	W =  -167.362 deg,	P =    -0.001 deg,	R =   120.301 deg
};
P[2889]{
   GP1:
	UF : 7, UT : 3,	CONFIG : 'F U T, 0, 0, 0',
	X =   278.445  mm,	Y =    78.332  mm,	Z =     0.000  mm,
	W =  -167.362 deg,	P =    -0.001 deg,	R =   120.301 deg
};
P[2890]{
   GP1:
	UF : 7, UT : 3,	CONFIG : 'F U T, 0, 0, 0',
	X =   278.445  mm,	Y =    78.332  mm,	Z =     0.000  mm,
	W =  -167.362 deg,	P =    -0.001 deg,	R =   120.301 deg
};
P[2891]{
   GP1:
	UF : 7, UT : 3,	CONFIG : 'F U T, 0, 0, 0',
	X =   278.445  mm,	Y =    78.332  mm,	Z =     0.000  mm,
	W =  -167.362 deg,	P =    -0.001 deg,	R =   120.301 deg
};
P[2892]{
   GP1:
	UF : 7, UT : 3,	CONFIG : 'F U T, 0, 0, 0',
	X =   272.605  mm,	Y =    96.720  mm,	Z =     0.001  mm,
	W =  -167.361 deg,	P =    -0.001 deg,	R =   124.584 deg
};
P[2893]{
   GP1:
	UF : 7, UT : 3,	CONFIG : 'F U T, 0, 0, 0',
	X =   265.154  mm,	Y =   115.600  mm,	Z =     0.001  mm,
	W =  -167.361 deg,	P =     0.000 deg,	R =   128.604 deg
};
P[2894]{
   GP1:
	UF : 7, UT : 3,	CONFIG : 'F U T, 0, 0, 0',
	X =   256.399  mm,	Y =   133.902  mm,	Z =     0.002  mm,
	W =  -167.361 deg,	P =     0.000 deg,	R =   132.625 deg
};
P[2895]{
   GP1:
	UF : 7, UT : 3,	CONFIG : 'F U T, 0, 0, 0',
	X =   246.387  mm,	Y =   151.536  mm,	Z =     0.001  mm,
	W =  -167.360 deg,	P =     0.000 deg,	R =   136.648 deg
};
P[2896]{
   GP1:
	UF : 7, UT : 3,	CONFIG : 'F U T, 0, 0, 0',
	X =   234.864  mm,	Y =   168.850  mm,	Z =     0.000  mm,
	W =  -167.359 deg,	P =     0.001 deg,	R =   140.583 deg
};
P[2897]{
   GP1:
	UF : 7, UT : 3,	CONFIG : 'F U T, 0, 0, 0',
	X =   234.864  mm,	Y =   168.850  mm,	Z =     0.000  mm,
	W =  -167.359 deg,	P =     0.001 deg,	R =   140.583 deg
};
P[2898]{
   GP1:
	UF : 7, UT : 3,	CONFIG : 'F U T, 0, 0, 0',
	X =   234.864  mm,	Y =   168.850  mm,	Z =     0.000  mm,
	W =  -167.359 deg,	P =     0.001 deg,	R =   140.583 deg
};
P[2899]{
   GP1:
	UF : 7, UT : 3,	CONFIG : 'F U T, 0, 0, 0',
	X =   234.864  mm,	Y =   168.850  mm,	Z =     0.000  mm,
	W =  -167.359 deg,	P =     0.001 deg,	R =   140.583 deg
};
P[2900]{
   GP1:
	UF : 7, UT : 3,	CONFIG : 'F U T, 0, 0, 0',
	X =   216.882  mm,	Y =   191.391  mm,	Z =     0.000  mm,
	W =  -167.361 deg,	P =    -0.002 deg,	R =   146.469 deg
};
P[2901]{
   GP1:
	UF : 7, UT : 3,	CONFIG : 'F U T, 0, 0, 0',
	X =   216.882  mm,	Y =   191.391  mm,	Z =     0.000  mm,
	W =  -167.361 deg,	P =    -0.002 deg,	R =   146.469 deg
};
P[2902]{
   GP1:
	UF : 7, UT : 3,	CONFIG : 'F U T, 0, 0, 0',
	X =   216.882  mm,	Y =   191.391  mm,	Z =     0.000  mm,
	W =  -167.361 deg,	P =    -0.002 deg,	R =   146.469 deg
};
P[2903]{
   GP1:
	UF : 7, UT : 3,	CONFIG : 'F U T, 0, 0, 0',
	X =   216.882  mm,	Y =   191.391  mm,	Z =     0.000  mm,
	W =  -167.361 deg,	P =    -0.002 deg,	R =   146.469 deg
};
P[2904]{
   GP1:
	UF : 7, UT : 3,	CONFIG : 'F U T, 0, 0, 0',
	X =   203.003  mm,	Y =   206.059  mm,	Z =     0.001  mm,
	W =  -167.361 deg,	P =    -0.002 deg,	R =   150.475 deg
};
P[2905]{
   GP1:
	UF : 7, UT : 3,	CONFIG : 'F U T, 0, 0, 0',
	X =   188.133  mm,	Y =   219.721  mm,	Z =     0.001  mm,
	W =  -167.360 deg,	P =    -0.001 deg,	R =   154.481 deg
};
P[2906]{
   GP1:
	UF : 7, UT : 3,	CONFIG : 'F U T, 0, 0, 0',
	X =   172.345  mm,	Y =   232.311  mm,	Z =     0.001  mm,
	W =  -167.360 deg,	P =     0.000 deg,	R =   158.487 deg
};
P[2907]{
   GP1:
	UF : 7, UT : 3,	CONFIG : 'F U T, 0, 0, 0',
	X =   155.715  mm,	Y =   243.767  mm,	Z =     0.001  mm,
	W =  -167.359 deg,	P =     0.000 deg,	R =   162.492 deg
};
P[2908]{
   GP1:
	UF : 7, UT : 3,	CONFIG : 'F U T, 0, 0, 0',
	X =   138.327  mm,	Y =   254.033  mm,	Z =     0.000  mm,
	W =  -167.359 deg,	P =     0.001 deg,	R =   166.498 deg
};
P[2909]{
   GP1:
	UF : 7, UT : 3,	CONFIG : 'F U T, 0, 0, 0',
	X =   138.327  mm,	Y =   254.033  mm,	Z =     0.000  mm,
	W =  -167.359 deg,	P =     0.001 deg,	R =   166.498 deg
};
P[2910]{
   GP1:
	UF : 7, UT : 3,	CONFIG : 'F U T, 0, 0, 0',
	X =   138.327  mm,	Y =   254.033  mm,	Z =     0.000  mm,
	W =  -167.359 deg,	P =     0.001 deg,	R =   166.498 deg
};
P[2911]{
   GP1:
	UF : 7, UT : 3,	CONFIG : 'F U T, 0, 0, 0',
	X =   138.327  mm,	Y =   254.033  mm,	Z =     0.000  mm,
	W =  -167.359 deg,	P =     0.001 deg,	R =   166.498 deg
};
P[2912]{
   GP1:
	UF : 7, UT : 3,	CONFIG : 'F U T, 0, 0, 0',
	X =   112.342  mm,	Y =   266.562  mm,	Z =     0.000  mm,
	W =  -167.361 deg,	P =    -0.002 deg,	R =   172.748 deg
};
P[2913]{
   GP1:
	UF : 7, UT : 3,	CONFIG : 'F U T, 0, 0, 0',
	X =   112.342  mm,	Y =   266.562  mm,	Z =     0.000  mm,
	W =  -167.361 deg,	P =    -0.002 deg,	R =   172.748 deg
};
P[2914]{
   GP1:
	UF : 7, UT : 3,	CONFIG : 'F U T, 0, 0, 0',
	X =   112.342  mm,	Y =   266.562  mm,	Z =     0.000  mm,
	W =  -167.361 deg,	P =    -0.002 deg,	R =   172.748 deg
};
P[2915]{
   GP1:
	UF : 7, UT : 3,	CONFIG : 'F U T, 0, 0, 0',
	X =   112.342  mm,	Y =   266.562  mm,	Z =     0.000  mm,
	W =  -167.361 deg,	P =    -0.002 deg,	R =   172.748 deg
};
P[2916]{
   GP1:
	UF : 7, UT : 3,	CONFIG : 'F U T, 0, 0, 0',
	X =    91.881  mm,	Y =   274.273  mm,	Z =     0.001  mm,
	W =  -167.361 deg,	P =    -0.001 deg,	R =   176.495 deg
};
P[2917]{
   GP1:
	UF : 7, UT : 3,	CONFIG : 'F U T, 0, 0, 0',
	X =    72.938  mm,	Y =   279.908  mm,	Z =     0.001  mm,
	W =  -167.361 deg,	P =    -0.001 deg,	R =  -179.569 deg
};
P[2918]{
   GP1:
	UF : 7, UT : 3,	CONFIG : 'F U T, 0, 0, 0',
	X =    53.633  mm,	Y =   284.242  mm,	Z =     0.001  mm,
	W =  -167.361 deg,	P =     0.000 deg,	R =  -175.638 deg
};
P[2919]{
   GP1:
	UF : 7, UT : 3,	CONFIG : 'F U T, 0, 0, 0',
	X =    34.061  mm,	Y =   287.246  mm,	Z =     0.001  mm,
	W =  -167.360 deg,	P =     0.000 deg,	R =  -171.710 deg
};
P[2920]{
   GP1:
	UF : 7, UT : 3,	CONFIG : 'F U T, 0, 0, 0',
	X =    14.416  mm,	Y =   288.897  mm,	Z =     0.000  mm,
	W =  -167.360 deg,	P =     0.001 deg,	R =  -167.766 deg
};
P[2921]{
   GP1:
	UF : 7, UT : 3,	CONFIG : 'F U T, 0, 0, 0',
	X =    14.416  mm,	Y =   288.897  mm,	Z =     0.000  mm,
	W =  -167.360 deg,	P =     0.001 deg,	R =  -167.766 deg
};
P[2922]{
   GP1:
	UF : 7, UT : 3,	CONFIG : 'F U T, 0, 0, 0',
	X =    14.416  mm,	Y =   288.897  mm,	Z =     0.000  mm,
	W =  -167.360 deg,	P =     0.001 deg,	R =  -167.766 deg
};
P[2923]{
   GP1:
	UF : 7, UT : 3,	CONFIG : 'F U T, 0, 0, 0',
	X =    14.416  mm,	Y =   288.897  mm,	Z =     0.000  mm,
	W =  -167.360 deg,	P =     0.001 deg,	R =  -167.766 deg
};
P[2924]{
   GP1:
	UF : 7, UT : 3,	CONFIG : 'F U T, 0, 0, 0',
	X =   -14.416  mm,	Y =   288.897  mm,	Z =     0.000  mm,
	W =  -167.360 deg,	P =    -0.003 deg,	R =  -162.071 deg
};
P[2925]{
   GP1:
	UF : 7, UT : 3,	CONFIG : 'F U T, 0, 0, 0',
	X =   -14.416  mm,	Y =   288.897  mm,	Z =     0.000  mm,
	W =  -167.360 deg,	P =    -0.003 deg,	R =  -162.071 deg
};
P[2926]{
   GP1:
	UF : 7, UT : 3,	CONFIG : 'F U T, 0, 0, 0',
	X =   -14.416  mm,	Y =   288.897  mm,	Z =     0.000  mm,
	W =  -167.360 deg,	P =    -0.003 deg,	R =  -162.071 deg
};
P[2927]{
   GP1:
	UF : 7, UT : 3,	CONFIG : 'F U T, 0, 0, 0',
	X =   -14.416  mm,	Y =   288.897  mm,	Z =     0.000  mm,
	W =  -167.360 deg,	P =    -0.003 deg,	R =  -162.071 deg
};
P[2928]{
   GP1:
	UF : 7, UT : 3,	CONFIG : 'F U T, 0, 0, 0',
	X =   -34.138  mm,	Y =   287.238  mm,	Z =     0.001  mm,
	W =  -167.359 deg,	P =    -0.001 deg,	R =  -158.155 deg
};
P[2929]{
   GP1:
	UF : 7, UT : 3,	CONFIG : 'F U T, 0, 0, 0',
	X =   -53.719  mm,	Y =   284.226  mm,	Z =     0.002  mm,
	W =  -167.358 deg,	P =     0.000 deg,	R =  -154.243 deg
};
P[2930]{
   GP1:
	UF : 7, UT : 3,	CONFIG : 'F U T, 0, 0, 0',
	X =   -73.012  mm,	Y =   279.888  mm,	Z =     0.002  mm,
	W =  -167.356 deg,	P =     0.001 deg,	R =  -150.325 deg
};
P[2931]{
   GP1:
	UF : 7, UT : 3,	CONFIG : 'F U T, 0, 0, 0',
	X =   -91.931  mm,	Y =   274.255  mm,	Z =     0.002  mm,
	W =  -167.354 deg,	P =     0.002 deg,	R =  -146.400 deg
};
P[2932]{
   GP1:
	UF : 7, UT : 3,	CONFIG : 'F U T, 0, 0, 0',
	X =  -112.342  mm,	Y =   266.562  mm,	Z =     0.000  mm,
	W =  -167.352 deg,	P =     0.002 deg,	R =  -142.645 deg
};
P[2933]{
   GP1:
	UF : 7, UT : 3,	CONFIG : 'F U T, 0, 0, 0',
	X =  -112.342  mm,	Y =   266.562  mm,	Z =     0.000  mm,
	W =  -167.352 deg,	P =     0.002 deg,	R =  -142.645 deg
};
P[2934]{
   GP1:
	UF : 7, UT : 3,	CONFIG : 'F U T, 0, 0, 0',
	X =  -112.342  mm,	Y =   266.562  mm,	Z =     0.000  mm,
	W =  -167.352 deg,	P =     0.002 deg,	R =  -142.645 deg
};
P[2935]{
   GP1:
	UF : 7, UT : 3,	CONFIG : 'F U T, 0, 0, 0',
	X =  -112.342  mm,	Y =   266.562  mm,	Z =     0.000  mm,
	W =  -167.352 deg,	P =     0.002 deg,	R =  -142.645 deg
};
P[2936]{
   GP1:
	UF : 7, UT : 3,	CONFIG : 'F U T, 0, 0, 0',
	X =  -138.327  mm,	Y =   254.033  mm,	Z =     0.000  mm,
	W =  -167.342 deg,	P =    -0.019 deg,	R =  -136.890 deg
};
P[2937]{
   GP1:
	UF : 7, UT : 3,	CONFIG : 'F U T, 0, 0, 0',
	X =  -138.327  mm,	Y =   254.033  mm,	Z =     0.000  mm,
	W =  -167.342 deg,	P =    -0.019 deg,	R =  -136.890 deg
};
P[2938]{
   GP1:
	UF : 7, UT : 3,	CONFIG : 'F U T, 0, 0, 0',
	X =  -138.327  mm,	Y =   254.033  mm,	Z =     0.000  mm,
	W =  -167.342 deg,	P =    -0.019 deg,	R =  -136.890 deg
};
P[2939]{
   GP1:
	UF : 7, UT : 3,	CONFIG : 'F U T, 0, 0, 0',
	X =  -138.327  mm,	Y =   254.033  mm,	Z =     0.000  mm,
	W =  -167.342 deg,	P =    -0.019 deg,	R =  -136.890 deg
};
P[2940]{
   GP1:
	UF : 7, UT : 3,	CONFIG : 'F U T, 0, 0, 0',
	X =  -150.066  mm,	Y =   247.282  mm,	Z =     0.005  mm,
	W =  -167.352 deg,	P =    -0.024 deg,	R =  -133.674 deg
};
P[2941]{
   GP1:
	UF : 7, UT : 3,	CONFIG : 'F U T, 0, 0, 0',
	X =  -162.485  mm,	Y =   239.322  mm,	Z =     0.016  mm,
	W =  -167.364 deg,	P =    -0.028 deg,	R =  -130.774 deg
};
P[2942]{
   GP1:
	UF : 7, UT : 3,	CONFIG : 'F U T, 0, 0, 0',
	X =  -174.433  mm,	Y =   230.744  mm,	Z =     0.026  mm,
	W =  -167.376 deg,	P =    -0.032 deg,	R =  -127.865 deg
};
P[2943]{
   GP1:
	UF : 7, UT : 3,	CONFIG : 'F U T, 0, 0, 0',
	X =  -187.272  mm,	Y =   220.459  mm,	Z =     0.032  mm,
	W =  -167.361 deg,	P =     0.001 deg,	R =  -124.599 deg
};
P[2944]{
   GP1:
	UF : 7, UT : 3,	CONFIG : 'F U T, 0, 0, 0',
	X =  -199.499  mm,	Y =   209.447  mm,	Z =     0.028  mm,
	W =  -167.343 deg,	P =     0.031 deg,	R =  -121.336 deg
};
P[2945]{
   GP1:
	UF : 7, UT : 3,	CONFIG : 'F U T, 0, 0, 0',
	X =  -208.545  mm,	Y =   200.442  mm,	Z =     0.017  mm,
	W =  -167.261 deg,	P =     0.037 deg,	R =  -118.804 deg
};
P[2946]{
   GP1:
	UF : 7, UT : 3,	CONFIG : 'F U T, 0, 0, 0',
	X =  -216.882  mm,	Y =   191.391  mm,	Z =     0.000  mm,
	W =  -167.182 deg,	P =     0.034 deg,	R =  -116.167 deg
};
P[2947]{
   GP1:
	UF : 7, UT : 3,	CONFIG : 'F U T, 0, 0, 0',
	X =  -216.882  mm,	Y =   191.391  mm,	Z =     0.000  mm,
	W =  -167.182 deg,	P =     0.034 deg,	R =  -116.167 deg
};
P[2948]{
   GP1:
	UF : 7, UT : 3,	CONFIG : 'F U T, 0, 0, 0',
	X =  -216.882  mm,	Y =   191.391  mm,	Z =     0.000  mm,
	W =  -167.182 deg,	P =     0.034 deg,	R =  -116.167 deg
};
P[2949]{
   GP1:
	UF : 7, UT : 3,	CONFIG : 'F U T, 0, 0, 0',
	X =  -216.882  mm,	Y =   191.391  mm,	Z =     0.000  mm,
	W =  -167.182 deg,	P =     0.034 deg,	R =  -116.167 deg
};
P[2950]{
   GP1:
	UF : 7, UT : 3,	CONFIG : 'F U T, 0, 0, 0',
	X =  -234.864  mm,	Y =   168.850  mm,	Z =     0.000  mm,
	W =  -167.097 deg,	P =    -0.235 deg,	R =  -110.476 deg
};
P[2951]{
   GP1:
	UF : 7, UT : 3,	CONFIG : 'F U T, 0, 0, 0',
	X =  -234.864  mm,	Y =   168.850  mm,	Z =     0.000  mm,
	W =  -167.097 deg,	P =    -0.235 deg,	R =  -110.476 deg
};
P[2952]{
   GP1:
	UF : 7, UT : 3,	CONFIG : 'F U T, 0, 0, 0',
	X =  -234.864  mm,	Y =   168.850  mm,	Z =     0.000  mm,
	W =  -167.097 deg,	P =    -0.235 deg,	R =  -110.476 deg
};
P[2953]{
   GP1:
	UF : 7, UT : 3,	CONFIG : 'F U T, 0, 0, 0',
	X =  -234.864  mm,	Y =   168.850  mm,	Z =     0.000  mm,
	W =  -167.097 deg,	P =    -0.235 deg,	R =  -110.476 deg
};
P[2954]{
   GP1:
	UF : 7, UT : 3,	CONFIG : 'F U T, 0, 0, 0',
	X =  -241.066  mm,	Y =   159.864  mm,	Z =     0.043  mm,
	W =  -167.290 deg,	P =    -0.308 deg,	R =  -108.496 deg
};
P[2955]{
   GP1:
	UF : 7, UT : 3,	CONFIG : 'F U T, 0, 0, 0',
	X =  -248.977  mm,	Y =   147.242  mm,	Z =     0.116  mm,
	W =  -167.654 deg,	P =    -0.189 deg,	R =  -105.549 deg
};
P[2956]{
   GP1:
	UF : 7, UT : 3,	CONFIG : 'F U T, 0, 0, 0',
	X =  -255.396  mm,	Y =   135.803  mm,	Z =     0.159  mm,
	W =  -167.849 deg,	P =     0.033 deg,	R =  -102.948 deg
};
P[2957]{
   GP1:
	UF : 7, UT : 3,	CONFIG : 'F U T, 0, 0, 0',
	X =  -260.804  mm,	Y =   125.101  mm,	Z =     0.156  mm,
	W =  -167.842 deg,	P =     0.260 deg,	R =  -100.577 deg
};
P[2958]{
   GP1:
	UF : 7, UT : 3,	CONFIG : 'F U T, 0, 0, 0',
	X =  -269.129  mm,	Y =   106.023  mm,	Z =     0.064  mm,
	W =  -167.476 deg,	P =     0.308 deg,	R =   -96.448 deg
};
P[2959]{
   GP1:
	UF : 7, UT : 3,	CONFIG : 'F U T, 0, 0, 0',
	X =  -273.782  mm,	Y =    93.358  mm,	Z =     0.017  mm,
	W =  -167.326 deg,	P =     0.122 deg,	R =   -93.774 deg
};
P[2960]{
   GP1:
	UF : 7, UT : 3,	CONFIG : 'F U T, 0, 0, 0',
	X =  -278.445  mm,	Y =    78.332  mm,	Z =     0.000  mm,
	W =  -167.321 deg,	P =     0.009 deg,	R =   -90.279 deg
};
P[2961]{
   GP1:
	UF : 7, UT : 3,	CONFIG : 'F U T, 0, 0, 0',
	X =  -278.445  mm,	Y =    78.332  mm,	Z =     0.000  mm,
	W =  -167.321 deg,	P =     0.009 deg,	R =   -90.279 deg
};
P[2962]{
   GP1:
	UF : 7, UT : 3,	CONFIG : 'F U T, 0, 0, 0',
	X =  -278.445  mm,	Y =    78.332  mm,	Z =     0.000  mm,
	W =  -167.321 deg,	P =     0.009 deg,	R =   -90.279 deg
};
P[2963]{
   GP1:
	UF : 7, UT : 3,	CONFIG : 'F U T, 0, 0, 0',
	X =  -278.445  mm,	Y =    78.332  mm,	Z =     0.000  mm,
	W =  -167.321 deg,	P =     0.009 deg,	R =   -90.279 deg
};
P[2964]{
   GP1:
	UF : 7, UT : 3,	CONFIG : 'F U T, 0, 1, 0',
	X =  -284.871  mm,	Y =    50.219  mm,	Z =     0.000  mm,
	W =  -167.355 deg,	P =    -0.008 deg,	R =   -84.578 deg
};
P[2965]{
   GP1:
	UF : 7, UT : 3,	CONFIG : 'F U T, 0, 1, 0',
	X =  -284.871  mm,	Y =    50.219  mm,	Z =     0.000  mm,
	W =  -167.355 deg,	P =    -0.008 deg,	R =   -84.578 deg
};
P[2966]{
   GP1:
	UF : 7, UT : 3,	CONFIG : 'F U T, 0, 1, 0',
	X =  -284.871  mm,	Y =    50.219  mm,	Z =     0.000  mm,
	W =  -167.355 deg,	P =    -0.008 deg,	R =   -84.578 deg
};
P[2967]{
   GP1:
	UF : 7, UT : 3,	CONFIG : 'F U T, 0, 1, 0',
	X =  -284.871  mm,	Y =    50.219  mm,	Z =     0.000  mm,
	W =  -167.355 deg,	P =    -0.008 deg,	R =   -84.578 deg
};
P[2968]{
   GP1:
	UF : 7, UT : 3,	CONFIG : 'F U T, 0, 1, 0',
	X =  -287.321  mm,	Y =    33.420  mm,	Z =     0.001  mm,
	W =  -167.358 deg,	P =    -0.004 deg,	R =   -81.599 deg
};
P[2969]{
   GP1:
	UF : 7, UT : 3,	CONFIG : 'F U T, 0, 1, 0',
	X =  -288.718  mm,	Y =    17.699  mm,	Z =     0.001  mm,
	W =  -167.360 deg,	P =     0.000 deg,	R =   -78.468 deg
};
P[2970]{
   GP1:
	UF : 7, UT : 3,	CONFIG : 'F U T, 0, 1, 0',
	X =  -289.270  mm,	Y =     0.000  mm,	Z =     0.000  mm,
	W =  -167.362 deg,	P =     0.004 deg,	R =   -75.519 deg
};
P[2971]{
   GP1:
	UF : 7, UT : 3,	CONFIG : 'F U T, 0, 1, 0',
	X =  -289.270  mm,	Y =     0.000  mm,	Z =     0.000  mm,
	W =  -167.362 deg,	P =     0.004 deg,	R =   -75.519 deg
};
P[2972]{
   GP1:
	UF : 7, UT : 3,	CONFIG : 'F U T, 0, 1, 0',
	X =  -289.270  mm,	Y =     0.000  mm,	Z =     0.000  mm,
	W =  -167.362 deg,	P =     0.004 deg,	R =   -75.519 deg
};
P[2973]{
   GP1:
	UF : 7, UT : 3,	CONFIG : 'F U T, 0, 1, 0',
	X =  -289.270  mm,	Y =     0.000  mm,	Z =     0.000  mm,
	W =  -167.362 deg,	P =     0.004 deg,	R =   -75.519 deg
};
P[2974]{
   GP1:
	UF : 7, UT : 3,	CONFIG : 'F U T, 0, 1, 0',
	X =  -286.136  mm,	Y =     0.000  mm,	Z =     0.000  mm,
	W =  -167.363 deg,	P =     0.004 deg,	R =   -75.540 deg
};
P[2975]{
   GP1:
	UF : 7, UT : 3,	CONFIG : 'F U T, 0, 1, 0',
	X =  -286.136  mm,	Y =     0.000  mm,	Z =     0.000  mm,
	W =  -167.363 deg,	P =     0.004 deg,	R =   -75.540 deg
};
P[2976]{
   GP1:
	UF : 7, UT : 3,	CONFIG : 'F U T, 0, 1, 0',
	X =  -286.136  mm,	Y =     0.000  mm,	Z =     0.000  mm,
	W =  -167.363 deg,	P =     0.004 deg,	R =   -75.540 deg
};
P[2977]{
   GP1:
	UF : 7, UT : 3,	CONFIG : 'F U T, 0, 1, 0',
	X =  -286.136  mm,	Y =     0.000  mm,	Z =     0.000  mm,
	W =  -167.363 deg,	P =     0.004 deg,	R =   -75.540 deg
};
P[2978]{
   GP1:
	UF : 7, UT : 3,	CONFIG : 'F U T, 0, 1, 0',
	X =  -285.285  mm,	Y =    21.849  mm,	Z =     0.001  mm,
	W =  -167.358 deg,	P =     0.000 deg,	R =   -79.336 deg
};
P[2979]{
   GP1:
	UF : 7, UT : 3,	CONFIG : 'F U T, 0, 1, 0',
	X =  -283.088  mm,	Y =    41.562  mm,	Z =     0.001  mm,
	W =  -167.354 deg,	P =    -0.003 deg,	R =   -83.290 deg
};
P[2980]{
   GP1:
	UF : 7, UT : 3,	CONFIG : 'F U T, 0, 0, 0',
	X =  -279.677  mm,	Y =    60.374  mm,	Z =     0.000  mm,
	W =  -167.350 deg,	P =    -0.005 deg,	R =   -87.604 deg
};
P[2981]{
   GP1:
	UF : 7, UT : 3,	CONFIG : 'F U T, 0, 0, 0',
	X =  -275.294  mm,	Y =    77.973  mm,	Z =     0.002  mm,
	W =  -167.340 deg,	P =     0.036 deg,	R =   -90.757 deg
};
P[2982]{
   GP1:
	UF : 7, UT : 3,	CONFIG : 'F U T, 0, 0, 0',
	X =  -271.856  mm,	Y =    89.226  mm,	Z =     0.011  mm,
	W =  -167.339 deg,	P =     0.076 deg,	R =   -93.116 deg
};
P[2983]{
   GP1:
	UF : 7, UT : 3,	CONFIG : 'F U T, 0, 0, 0',
	X =  -266.629  mm,	Y =   103.805  mm,	Z =     0.050  mm,
	W =  -167.469 deg,	P =     0.237 deg,	R =   -96.222 deg
};
P[2984]{
   GP1:
	UF : 7, UT : 3,	CONFIG : 'F U T, 0, 0, 0',
	X =  -261.798  mm,	Y =   115.450  mm,	Z =     0.101  mm,
	W =  -167.689 deg,	P =     0.319 deg,	R =   -98.743 deg
};
P[2985]{
   GP1:
	UF : 7, UT : 3,	CONFIG : 'F U T, 0, 0, 0',
	X =  -256.793  mm,	Y =   126.192  mm,	Z =     0.132  mm,
	W =  -167.832 deg,	P =     0.202 deg,	R =  -101.119 deg
};
P[2986]{
   GP1:
	UF : 7, UT : 3,	CONFIG : 'F U T, 0, 0, 0',
	X =  -250.756  mm,	Y =   137.801  mm,	Z =     0.128  mm,
	W =  -167.798 deg,	P =     0.001 deg,	R =  -103.739 deg
};
P[2987]{
   GP1:
	UF : 7, UT : 3,	CONFIG : 'F U T, 0, 0, 0',
	X =  -242.629  mm,	Y =   151.646  mm,	Z =     0.077  mm,
	W =  -167.535 deg,	P =    -0.178 deg,	R =  -106.947 deg
};
P[2988]{
   GP1:
	UF : 7, UT : 3,	CONFIG : 'F U T, 0, 0, 0',
	X =  -233.847  mm,	Y =   164.876  mm,	Z =     0.022  mm,
	W =  -167.222 deg,	P =    -0.201 deg,	R =  -110.133 deg
};
P[2989]{
   GP1:
	UF : 7, UT : 3,	CONFIG : 'F U T, 0, 0, 0',
	X =  -221.510  mm,	Y =   181.125  mm,	Z =     0.000  mm,
	W =  -167.152 deg,	P =    -0.034 deg,	R =  -114.137 deg
};
P[2990]{
   GP1:
	UF : 7, UT : 3,	CONFIG : 'F U T, 0, 0, 0',
	X =  -207.946  mm,	Y =   196.530  mm,	Z =     0.018  mm,
	W =  -167.290 deg,	P =     0.036 deg,	R =  -118.342 deg
};
P[2991]{
   GP1:
	UF : 7, UT : 3,	CONFIG : 'F U T, 0, 0, 0',
	X =  -198.736  mm,	Y =   205.842  mm,	Z =     0.028  mm,
	W =  -167.341 deg,	P =     0.025 deg,	R =  -120.961 deg
};
P[2992]{
   GP1:
	UF : 7, UT : 3,	CONFIG : 'F U T, 0, 0, 0',
	X =  -189.097  mm,	Y =   214.731  mm,	Z =     0.031  mm,
	W =  -167.391 deg,	P =     0.010 deg,	R =  -123.576 deg
};
P[2993]{
   GP1:
	UF : 7, UT : 3,	CONFIG : 'F U T, 0, 0, 0',
	X =  -174.298  mm,	Y =   226.904  mm,	Z =     0.027  mm,
	W =  -167.380 deg,	P =    -0.016 deg,	R =  -127.397 deg
};
P[2994]{
   GP1:
	UF : 7, UT : 3,	CONFIG : 'F U T, 0, 0, 0',
	X =  -158.838  mm,	Y =   237.981  mm,	Z =     0.015  mm,
	W =  -167.365 deg,	P =    -0.041 deg,	R =  -131.246 deg
};
P[2995]{
   GP1:
	UF : 7, UT : 3,	CONFIG : 'F U T, 0, 0, 0',
	X =  -143.540  mm,	Y =   247.511  mm,	Z =     0.004  mm,
	W =  -167.354 deg,	P =    -0.025 deg,	R =  -134.853 deg
};
P[2996]{
   GP1:
	UF : 7, UT : 3,	CONFIG : 'F U T, 0, 0, 0',
	X =  -127.238  mm,	Y =   256.279  mm,	Z =     0.000  mm,
	W =  -167.345 deg,	P =    -0.007 deg,	R =  -138.815 deg
};
P[2997]{
   GP1:
	UF : 7, UT : 3,	CONFIG : 'F U T, 0, 0, 0',
	X =  -121.064  mm,	Y =   259.248  mm,	Z =     0.000  mm,
	W =  -167.348 deg,	P =    -0.003 deg,	R =  -139.601 deg
};
P[2998]{
   GP1:
	UF : 7, UT : 3,	CONFIG : 'F U T, 0, 0, 0',
	X =  -102.132  mm,	Y =   267.271  mm,	Z =     0.001  mm,
	W =  -167.350 deg,	P =    -0.002 deg,	R =  -144.019 deg
};
P[2999]{
   GP1:
	UF : 7, UT : 3,	CONFIG : 'F U T, 0, 0, 0',
	X =   -82.792  mm,	Y =   273.885  mm,	Z =     0.002  mm,
	W =  -167.352 deg,	P =    -0.001 deg,	R =  -148.116 deg
};
P[3000]{
   GP1:
	UF : 7, UT : 3,	CONFIG : 'F U T, 0, 0, 0',
	X =   -63.028  mm,	Y =   279.099  mm,	Z =     0.002  mm,
	W =  -167.354 deg,	P =    -0.001 deg,	R =  -152.214 deg
};
P[3001]{
   GP1:
	UF : 7, UT : 3,	CONFIG : 'F U T, 0, 0, 0',
	X =   -42.961  mm,	Y =   282.880  mm,	Z =     0.002  mm,
	W =  -167.356 deg,	P =    -0.001 deg,	R =  -156.318 deg
};
P[3002]{
   GP1:
	UF : 7, UT : 3,	CONFIG : 'F U T, 0, 0, 0',
	X =   -22.558  mm,	Y =   285.230  mm,	Z =     0.001  mm,
	W =  -167.358 deg,	P =    -0.001 deg,	R =  -160.398 deg
};
P[3003]{
   GP1:
	UF : 7, UT : 3,	CONFIG : 'F U T, 0, 0, 0',
	X =    -3.366  mm,	Y =   286.099  mm,	Z =     0.000  mm,
	W =  -167.359 deg,	P =    -0.002 deg,	R =  -164.890 deg
};
P[3004]{
   GP1:
	UF : 7, UT : 3,	CONFIG : 'F U T, 0, 0, 0',
	X =     3.366  mm,	Y =   286.099  mm,	Z =     0.000  mm,
	W =  -167.359 deg,	P =    -0.001 deg,	R =  -165.022 deg
};
P[3005]{
   GP1:
	UF : 7, UT : 3,	CONFIG : 'F U T, 0, 0, 0',
	X =    22.629  mm,	Y =   285.225  mm,	Z =     0.000  mm,
	W =  -167.360 deg,	P =    -0.001 deg,	R =  -169.504 deg
};
P[3006]{
   GP1:
	UF : 7, UT : 3,	CONFIG : 'F U T, 0, 0, 0',
	X =    43.004  mm,	Y =   282.874  mm,	Z =     0.001  mm,
	W =  -167.360 deg,	P =    -0.001 deg,	R =  -173.583 deg
};
P[3007]{
   GP1:
	UF : 7, UT : 3,	CONFIG : 'F U T, 0, 0, 0',
	X =    63.053  mm,	Y =   279.092  mm,	Z =     0.001  mm,
	W =  -167.360 deg,	P =    -0.001 deg,	R =  -177.684 deg
};
P[3008]{
   GP1:
	UF : 7, UT : 3,	CONFIG : 'F U T, 0, 0, 0',
	X =    82.799  mm,	Y =   273.884  mm,	Z =     0.001  mm,
	W =  -167.360 deg,	P =    -0.001 deg,	R =   178.219 deg
};
P[3009]{
   GP1:
	UF : 7, UT : 3,	CONFIG : 'F U T, 0, 0, 0',
	X =   102.079  mm,	Y =   267.291  mm,	Z =     0.000  mm,
	W =  -167.360 deg,	P =    -0.001 deg,	R =   174.112 deg
};
P[3010]{
   GP1:
	UF : 7, UT : 3,	CONFIG : 'F U T, 0, 0, 0',
	X =   121.064  mm,	Y =   259.248  mm,	Z =     0.000  mm,
	W =  -167.360 deg,	P =    -0.001 deg,	R =   169.708 deg
};
P[3011]{
   GP1:
	UF : 7, UT : 3,	CONFIG : 'F U T, 0, 0, 0',
	X =   127.238  mm,	Y =   256.279  mm,	Z =     0.000  mm,
	W =  -167.359 deg,	P =    -0.001 deg,	R =   168.918 deg
};
P[3012]{
   GP1:
	UF : 7, UT : 3,	CONFIG : 'F U T, 0, 0, 0',
	X =   145.093  mm,	Y =   246.608  mm,	Z =     0.001  mm,
	W =  -167.359 deg,	P =    -0.001 deg,	R =   164.591 deg
};
P[3013]{
   GP1:
	UF : 7, UT : 3,	CONFIG : 'F U T, 0, 0, 0',
	X =   161.798  mm,	Y =   235.991  mm,	Z =     0.002  mm,
	W =  -167.360 deg,	P =    -0.001 deg,	R =   160.620 deg
};
P[3014]{
   GP1:
	UF : 7, UT : 3,	CONFIG : 'F U T, 0, 0, 0',
	X =   177.733  mm,	Y =   224.223  mm,	Z =     0.002  mm,
	W =  -167.360 deg,	P =    -0.001 deg,	R =   156.651 deg
};
P[3015]{
   GP1:
	UF : 7, UT : 3,	CONFIG : 'F U T, 0, 0, 0',
	X =   192.823  mm,	Y =   211.389  mm,	Z =     0.001  mm,
	W =  -167.360 deg,	P =    -0.001 deg,	R =   152.684 deg
};
P[3016]{
   GP1:
	UF : 7, UT : 3,	CONFIG : 'F U T, 0, 0, 0',
	X =   206.992  mm,	Y =   197.536  mm,	Z =     0.001  mm,
	W =  -167.360 deg,	P =    -0.001 deg,	R =   148.717 deg
};
P[3017]{
   GP1:
	UF : 7, UT : 3,	CONFIG : 'F U T, 0, 0, 0',
	X =   221.510  mm,	Y =   181.125  mm,	Z =     0.000  mm,
	W =  -167.360 deg,	P =    -0.001 deg,	R =   144.241 deg
};
P[3018]{
   GP1:
	UF : 7, UT : 3,	CONFIG : 'F U T, 0, 0, 0',
	X =   225.844  mm,	Y =   175.682  mm,	Z =     0.000  mm,
	W =  -167.360 deg,	P =    -0.001 deg,	R =   143.097 deg
};
P[3019]{
   GP1:
	UF : 7, UT : 3,	CONFIG : 'F U T, 0, 0, 0',
	X =   238.160  mm,	Y =   158.575  mm,	Z =     0.001  mm,
	W =  -167.360 deg,	P =     0.000 deg,	R =   138.706 deg
};
P[3020]{
   GP1:
	UF : 7, UT : 3,	CONFIG : 'F U T, 0, 0, 0',
	X =   248.771  mm,	Y =   141.345  mm,	Z =     0.002  mm,
	W =  -167.361 deg,	P =     0.000 deg,	R =   134.679 deg
};
P[3021]{
   GP1:
	UF : 7, UT : 3,	CONFIG : 'F U T, 0, 0, 0',
	X =   258.085  mm,	Y =   123.529  mm,	Z =     0.002  mm,
	W =  -167.361 deg,	P =     0.000 deg,	R =   130.626 deg
};
P[3022]{
   GP1:
	UF : 7, UT : 3,	CONFIG : 'F U T, 0, 0, 0',
	X =   266.141  mm,	Y =   105.054  mm,	Z =     0.001  mm,
	W =  -167.361 deg,	P =     0.000 deg,	R =   126.583 deg
};
P[3023]{
   GP1:
	UF : 7, UT : 3,	CONFIG : 'F U T, 0, 0, 0',
	X =   272.900  mm,	Y =    85.972  mm,	Z =     0.000  mm,
	W =  -167.362 deg,	P =     0.000 deg,	R =   122.557 deg
};
P[3024]{
   GP1:
	UF : 7, UT : 3,	CONFIG : 'F U T, 0, 0, 0',
	X =   278.174  mm,	Y =    66.966  mm,	Z =     0.000  mm,
	W =  -167.362 deg,	P =    -0.001 deg,	R =   118.159 deg
};
P[3025]{
   GP1:
	UF : 7, UT : 3,	CONFIG : 'F U T, 0, 0, 0',
	X =   279.677  mm,	Y =    60.374  mm,	Z =     0.000  mm,
	W =  -167.362 deg,	P =     0.000 deg,	R =   117.729 deg
};
P[3026]{
   GP1:
	UF : 7, UT : 3,	CONFIG : 'F U T, 0, 0, 0',
	X =   283.077  mm,	Y =    41.630  mm,	Z =     0.000  mm,
	W =  -167.363 deg,	P =     0.000 deg,	R =   113.412 deg
};
P[3027]{
   GP1:
	UF : 7, UT : 3,	CONFIG : 'F U T, 0, 0, 0',
	X =   285.282  mm,	Y =    21.888  mm,	Z =     0.000  mm,
	W =  -167.363 deg,	P =    -0.001 deg,	R =   109.461 deg
};
P[3028]{
   GP1:
	UF : 7, UT : 3,	CONFIG : 'F U T, 0, 0, 0',
	X =   286.136  mm,	Y =     0.000  mm,	Z =     0.000  mm,
	W =  -167.364 deg,	P =    -0.001 deg,	R =   105.651 deg
};
P[3029]{
   GP1:
	UF : 7, UT : 3,	CONFIG : 'F U T, 0, 0, 0',
	X =   286.136  mm,	Y =     0.000  mm,	Z =     0.000  mm,
	W =  -167.364 deg,	P =    -0.001 deg,	R =   105.651 deg
};
P[3030]{
   GP1:
	UF : 7, UT : 3,	CONFIG : 'F U T, 0, 0, 0',
	X =   286.136  mm,	Y =     0.000  mm,	Z =     0.000  mm,
	W =  -167.364 deg,	P =    -0.001 deg,	R =   105.651 deg
};
P[3031]{
   GP1:
	UF : 7, UT : 3,	CONFIG : 'F U T, 0, 0, 0',
	X =   286.136  mm,	Y =     0.000  mm,	Z =     0.000  mm,
	W =  -167.364 deg,	P =    -0.001 deg,	R =   105.651 deg
};
P[3032]{
   GP1:
	UF : 7, UT : 3,	CONFIG : 'F U T, 0, 0, 0',
	X =   283.002  mm,	Y =     0.000  mm,	Z =     0.000  mm,
	W =  -167.364 deg,	P =    -0.001 deg,	R =   105.637 deg
};
P[3033]{
   GP1:
	UF : 7, UT : 3,	CONFIG : 'F U T, 0, 0, 0',
	X =   283.002  mm,	Y =     0.000  mm,	Z =     0.000  mm,
	W =  -167.364 deg,	P =    -0.001 deg,	R =   105.637 deg
};
P[3034]{
   GP1:
	UF : 7, UT : 3,	CONFIG : 'F U T, 0, 0, 0',
	X =   283.002  mm,	Y =     0.000  mm,	Z =     0.000  mm,
	W =  -167.364 deg,	P =    -0.001 deg,	R =   105.637 deg
};
P[3035]{
   GP1:
	UF : 7, UT : 3,	CONFIG : 'F U T, 0, 0, 0',
	X =   283.002  mm,	Y =     0.000  mm,	Z =     0.000  mm,
	W =  -167.364 deg,	P =    -0.001 deg,	R =   105.637 deg
};
P[3036]{
   GP1:
	UF : 7, UT : 3,	CONFIG : 'F U T, 0, 0, 0',
	X =   282.182  mm,	Y =    21.348  mm,	Z =     0.000  mm,
	W =  -167.363 deg,	P =    -0.001 deg,	R =   109.388 deg
};
P[3037]{
   GP1:
	UF : 7, UT : 3,	CONFIG : 'F U T, 0, 0, 0',
	X =   280.052  mm,	Y =    40.648  mm,	Z =     0.000  mm,
	W =  -167.363 deg,	P =    -0.001 deg,	R =   113.297 deg
};
P[3038]{
   GP1:
	UF : 7, UT : 3,	CONFIG : 'F U T, 0, 0, 0',
	X =   276.634  mm,	Y =    59.631  mm,	Z =     0.000  mm,
	W =  -167.363 deg,	P =    -0.001 deg,	R =   117.232 deg
};
P[3039]{
   GP1:
	UF : 7, UT : 3,	CONFIG : 'F U T, 0, 0, 0',
	X =   271.914  mm,	Y =    78.398  mm,	Z =     0.000  mm,
	W =  -167.363 deg,	P =     0.000 deg,	R =   121.154 deg
};
P[3040]{
   GP1:
	UF : 7, UT : 3,	CONFIG : 'F U T, 0, 0, 0',
	X =   265.908  mm,	Y =    96.839  mm,	Z =     0.001  mm,
	W =  -167.362 deg,	P =     0.000 deg,	R =   125.067 deg
};
P[3041]{
   GP1:
	UF : 7, UT : 3,	CONFIG : 'F U T, 0, 0, 0',
	X =   258.667  mm,	Y =   114.797  mm,	Z =     0.001  mm,
	W =  -167.362 deg,	P =    -0.001 deg,	R =   128.987 deg
};
P[3042]{
   GP1:
	UF : 7, UT : 3,	CONFIG : 'F U T, 0, 0, 0',
	X =   250.212  mm,	Y =   132.224  mm,	Z =     0.002  mm,
	W =  -167.362 deg,	P =    -0.001 deg,	R =   132.905 deg
};
P[3043]{
   GP1:
	UF : 7, UT : 3,	CONFIG : 'F U T, 0, 0, 0',
	X =   240.585  mm,	Y =   149.020  mm,	Z =     0.001  mm,
	W =  -167.361 deg,	P =    -0.001 deg,	R =   136.828 deg
};
P[3044]{
   GP1:
	UF : 7, UT : 3,	CONFIG : 'F U T, 0, 0, 0',
	X =   229.831  mm,	Y =   165.119  mm,	Z =     0.000  mm,
	W =  -167.361 deg,	P =    -0.001 deg,	R =   140.748 deg
};
P[3045]{
   GP1:
	UF : 7, UT : 3,	CONFIG : 'F U T, 0, 0, 0',
	X =   217.988  mm,	Y =   180.463  mm,	Z =     0.000  mm,
	W =  -167.361 deg,	P =    -0.001 deg,	R =   144.664 deg
};
P[3046]{
   GP1:
	UF : 7, UT : 3,	CONFIG : 'F U T, 0, 0, 0',
	X =   205.860  mm,	Y =   194.177  mm,	Z =     0.001  mm,
	W =  -167.361 deg,	P =    -0.001 deg,	R =   148.378 deg
};
P[3047]{
   GP1:
	UF : 7, UT : 3,	CONFIG : 'F U T, 0, 0, 0',
	X =   192.892  mm,	Y =   207.062  mm,	Z =     0.001  mm,
	W =  -167.361 deg,	P =    -0.001 deg,	R =   152.102 deg
};
P[3048]{
   GP1:
	UF : 7, UT : 3,	CONFIG : 'F U T, 0, 0, 0',
	X =   179.026  mm,	Y =   219.166  mm,	Z =     0.002  mm,
	W =  -167.362 deg,	P =    -0.001 deg,	R =   155.795 deg
};
P[3049]{
   GP1:
	UF : 7, UT : 3,	CONFIG : 'F U T, 0, 0, 0',
	X =   164.530  mm,	Y =   230.250  mm,	Z =     0.002  mm,
	W =  -167.362 deg,	P =    -0.001 deg,	R =   159.521 deg
};
P[3050]{
   GP1:
	UF : 7, UT : 3,	CONFIG : 'F U T, 0, 0, 0',
	X =   149.265  mm,	Y =   240.431  mm,	Z =     0.001  mm,
	W =  -167.362 deg,	P =    -0.001 deg,	R =   163.225 deg
};
P[3051]{
   GP1:
	UF : 7, UT : 3,	CONFIG : 'F U T, 0, 0, 0',
	X =   133.351  mm,	Y =   249.604  mm,	Z =     0.000  mm,
	W =  -167.362 deg,	P =    -0.001 deg,	R =   166.927 deg
};
P[3052]{
   GP1:
	UF : 7, UT : 3,	CONFIG : 'F U T, 0, 0, 0',
	X =   116.962  mm,	Y =   257.685  mm,	Z =     0.000  mm,
	W =  -167.363 deg,	P =    -0.001 deg,	R =   170.647 deg
};
P[3053]{
   GP1:
	UF : 7, UT : 3,	CONFIG : 'F U T, 0, 0, 0',
	X =   100.036  mm,	Y =   264.717  mm,	Z =     0.001  mm,
	W =  -167.363 deg,	P =    -0.001 deg,	R =   174.356 deg
};
P[3054]{
   GP1:
	UF : 7, UT : 3,	CONFIG : 'F U T, 0, 0, 0',
	X =    82.700  mm,	Y =   270.635  mm,	Z =     0.001  mm,
	W =  -167.363 deg,	P =    -0.001 deg,	R =   178.066 deg
};
P[3055]{
   GP1:
	UF : 7, UT : 3,	CONFIG : 'F U T, 0, 0, 0',
	X =    64.971  mm,	Y =   275.431  mm,	Z =     0.001  mm,
	W =  -167.363 deg,	P =     0.000 deg,	R =  -178.233 deg
};
P[3056]{
   GP1:
	UF : 7, UT : 3,	CONFIG : 'F U T, 0, 0, 0',
	X =    48.469  mm,	Y =   278.805  mm,	Z =     0.001  mm,
	W =  -167.363 deg,	P =     0.000 deg,	R =  -174.809 deg
};
P[3057]{
   GP1:
	UF : 7, UT : 3,	CONFIG : 'F U T, 0, 0, 0',
	X =    31.759  mm,	Y =   281.207  mm,	Z =     0.001  mm,
	W =  -167.362 deg,	P =     0.000 deg,	R =  -171.388 deg
};
P[3058]{
   GP1:
	UF : 7, UT : 3,	CONFIG : 'F U T, 0, 0, 0',
	X =    14.970  mm,	Y =   282.591  mm,	Z =     0.000  mm,
	W =  -167.362 deg,	P =     0.001 deg,	R =  -167.965 deg
};
P[3059]{
   GP1:
	UF : 7, UT : 3,	CONFIG : 'F U T, 0, 0, 0',
	X =    -1.898  mm,	Y =   282.985  mm,	Z =     0.000  mm,
	W =  -167.361 deg,	P =     0.001 deg,	R =  -164.545 deg
};
P[3060]{
   GP1:
	UF : 7, UT : 3,	CONFIG : 'F U T, 0, 0, 0',
	X =   -18.840  mm,	Y =   282.374  mm,	Z =     0.001  mm,
	W =  -167.361 deg,	P =     0.001 deg,	R =  -161.140 deg
};
P[3061]{
   GP1:
	UF : 7, UT : 3,	CONFIG : 'F U T, 0, 0, 0',
	X =   -35.609  mm,	Y =   280.737  mm,	Z =     0.001  mm,
	W =  -167.360 deg,	P =     0.001 deg,	R =  -157.712 deg
};
P[3062]{
   GP1:
	UF : 7, UT : 3,	CONFIG : 'F U T, 0, 0, 0',
	X =   -52.290  mm,	Y =   278.117  mm,	Z =     0.002  mm,
	W =  -167.360 deg,	P =     0.002 deg,	R =  -154.298 deg
};
P[3063]{
   GP1:
	UF : 7, UT : 3,	CONFIG : 'F U T, 0, 0, 0',
	X =   -68.791  mm,	Y =   274.500  mm,	Z =     0.002  mm,
	W =  -167.359 deg,	P =     0.002 deg,	R =  -150.884 deg
};
P[3064]{
   GP1:
	UF : 7, UT : 3,	CONFIG : 'F U T, 0, 0, 0',
	X =   -85.005  mm,	Y =   269.922  mm,	Z =     0.002  mm,
	W =  -167.358 deg,	P =     0.001 deg,	R =  -147.461 deg
};
P[3065]{
   GP1:
	UF : 7, UT : 3,	CONFIG : 'F U T, 0, 0, 0',
	X =  -100.964  mm,	Y =   264.364  mm,	Z =     0.002  mm,
	W =  -167.358 deg,	P =     0.001 deg,	R =  -144.048 deg
};
P[3066]{
   GP1:
	UF : 7, UT : 3,	CONFIG : 'F U T, 0, 0, 0',
	X =  -117.167  mm,	Y =   257.591  mm,	Z =     0.001  mm,
	W =  -167.357 deg,	P =    -0.010 deg,	R =  -140.501 deg
};
P[3067]{
   GP1:
	UF : 7, UT : 3,	CONFIG : 'F U T, 0, 0, 0',
	X =  -132.874  mm,	Y =   249.862  mm,	Z =     0.002  mm,
	W =  -167.358 deg,	P =    -0.021 deg,	R =  -136.942 deg
};
P[3068]{
   GP1:
	UF : 7, UT : 3,	CONFIG : 'F U T, 0, 0, 0',
	X =  -148.094  mm,	Y =   241.153  mm,	Z =     0.009  mm,
	W =  -167.360 deg,	P =    -0.033 deg,	R =  -133.389 deg
};
P[3069]{
   GP1:
	UF : 7, UT : 3,	CONFIG : 'F U T, 0, 0, 0',
	X =  -161.267  mm,	Y =   232.541  mm,	Z =     0.018  mm,
	W =  -167.380 deg,	P =    -0.020 deg,	R =  -130.218 deg
};
P[3070]{
   GP1:
	UF : 7, UT : 3,	CONFIG : 'F U T, 0, 0, 0',
	X =  -173.885  mm,	Y =   223.264  mm,	Z =     0.026  mm,
	W =  -167.398 deg,	P =    -0.005 deg,	R =  -127.030 deg
};
P[3071]{
   GP1:
	UF : 7, UT : 3,	CONFIG : 'F U T, 0, 0, 0',
	X =  -186.005  mm,	Y =   213.273  mm,	Z =     0.029  mm,
	W =  -167.414 deg,	P =     0.011 deg,	R =  -123.853 deg
};
P[3072]{
   GP1:
	UF : 7, UT : 3,	CONFIG : 'F U T, 0, 0, 0',
	X =  -197.905  mm,	Y =   202.278  mm,	Z =     0.026  mm,
	W =  -167.357 deg,	P =     0.020 deg,	R =  -120.574 deg
};
P[3073]{
   GP1:
	UF : 7, UT : 3,	CONFIG : 'F U T, 0, 0, 0',
	X =  -209.155  mm,	Y =   190.624  mm,	Z =     0.017  mm,
	W =  -167.299 deg,	P =     0.021 deg,	R =  -117.294 deg
};
P[3074]{
   GP1:
	UF : 7, UT : 3,	CONFIG : 'F U T, 0, 0, 0',
	X =  -216.516  mm,	Y =   182.214  mm,	Z =     0.011  mm,
	W =  -167.258 deg,	P =    -0.024 deg,	R =  -115.034 deg
};
P[3075]{
   GP1:
	UF : 7, UT : 3,	CONFIG : 'F U T, 0, 0, 0',
	X =  -223.534  mm,	Y =   173.540  mm,	Z =     0.011  mm,
	W =  -167.219 deg,	P =    -0.073 deg,	R =  -112.771 deg
};
P[3076]{
   GP1:
	UF : 7, UT : 3,	CONFIG : 'F U T, 0, 0, 0',
	X =  -231.947  mm,	Y =   162.114  mm,	Z =     0.032  mm,
	W =  -167.330 deg,	P =    -0.142 deg,	R =  -109.913 deg
};
P[3077]{
   GP1:
	UF : 7, UT : 3,	CONFIG : 'F U T, 0, 0, 0',
	X =  -243.096  mm,	Y =   144.873  mm,	Z =     0.085  mm,
	W =  -167.671 deg,	P =    -0.065 deg,	R =  -105.757 deg
};
P[3078]{
   GP1:
	UF : 7, UT : 3,	CONFIG : 'F U T, 0, 0, 0',
	X =  -250.599  mm,	Y =   131.482  mm,	Z =     0.109  mm,
	W =  -167.819 deg,	P =     0.102 deg,	R =  -102.633 deg
};
P[3079]{
   GP1:
	UF : 7, UT : 3,	CONFIG : 'F U T, 0, 0, 0',
	X =  -256.287  mm,	Y =   120.013  mm,	Z =     0.097  mm,
	W =  -167.762 deg,	P =     0.236 deg,	R =  -100.039 deg
};
P[3080]{
   GP1:
	UF : 7, UT : 3,	CONFIG : 'F U T, 0, 0, 0',
	X =  -261.363  mm,	Y =   108.511  mm,	Z =     0.060  mm,
	W =  -167.572 deg,	P =     0.248 deg,	R =   -97.495 deg
};
P[3081]{
   GP1:
	UF : 7, UT : 3,	CONFIG : 'F U T, 0, 0, 0',
	X =  -267.261  mm,	Y =    93.028  mm,	Z =     0.018  mm,
	W =  -167.381 deg,	P =     0.106 deg,	R =   -94.140 deg
};
P[3082]{
   GP1:
	UF : 7, UT : 3,	CONFIG : 'F U T, 0, 0, 0',
	X =  -273.326  mm,	Y =    73.320  mm,	Z =     0.002  mm,
	W =  -167.346 deg,	P =     0.008 deg,	R =   -89.966 deg
};
P[3083]{
   GP1:
	UF : 7, UT : 3,	CONFIG : 'F U T, 0, 1, 0',
	X =  -277.442  mm,	Y =    55.759  mm,	Z =     0.001  mm,
	W =  -167.350 deg,	P =     0.006 deg,	R =   -86.309 deg
};
P[3084]{
   GP1:
	UF : 7, UT : 3,	CONFIG : 'F U T, 0, 1, 0',
	X =  -280.436  mm,	Y =    37.961  mm,	Z =     0.001  mm,
	W =  -167.354 deg,	P =     0.005 deg,	R =   -82.655 deg
};
P[3085]{
   GP1:
	UF : 7, UT : 3,	CONFIG : 'F U T, 0, 1, 0',
	X =  -282.290  mm,	Y =    19.993  mm,	Z =     0.001  mm,
	W =  -167.358 deg,	P =     0.004 deg,	R =   -79.003 deg
};
P[3086]{
   GP1:
	UF : 7, UT : 3,	CONFIG : 'F U T, 0, 1, 0',
	X =  -283.002  mm,	Y =     0.000  mm,	Z =     0.000  mm,
	W =  -167.363 deg,	P =     0.003 deg,	R =   -75.524 deg
};
P[3087]{
   GP1:
	UF : 7, UT : 3,	CONFIG : 'F U T, 0, 1, 0',
	X =  -283.002  mm,	Y =     0.000  mm,	Z =     0.000  mm,
	W =  -167.363 deg,	P =     0.003 deg,	R =   -75.524 deg
};
P[3088]{
   GP1:
	UF : 7, UT : 3,	CONFIG : 'F U T, 0, 1, 0',
	X =  -283.002  mm,	Y =     0.000  mm,	Z =     0.000  mm,
	W =  -167.363 deg,	P =     0.003 deg,	R =   -75.524 deg
};
P[3089]{
   GP1:
	UF : 7, UT : 3,	CONFIG : 'F U T, 0, 1, 0',
	X =  -283.002  mm,	Y =     0.000  mm,	Z =     0.000  mm,
	W =  -167.363 deg,	P =     0.003 deg,	R =   -75.524 deg
};
P[3090]{
   GP1:
	UF : 7, UT : 3,	CONFIG : 'F U T, 0, 1, 0',
	X =  -279.868  mm,	Y =     0.000  mm,	Z =     0.000  mm,
	W =  -167.363 deg,	P =     0.003 deg,	R =   -75.545 deg
};
P[3091]{
   GP1:
	UF : 7, UT : 3,	CONFIG : 'F U T, 0, 1, 0',
	X =  -279.868  mm,	Y =     0.000  mm,	Z =     0.000  mm,
	W =  -167.363 deg,	P =     0.003 deg,	R =   -75.545 deg
};
P[3092]{
   GP1:
	UF : 7, UT : 3,	CONFIG : 'F U T, 0, 1, 0',
	X =  -279.868  mm,	Y =     0.000  mm,	Z =     0.000  mm,
	W =  -167.363 deg,	P =     0.003 deg,	R =   -75.545 deg
};
P[3093]{
   GP1:
	UF : 7, UT : 3,	CONFIG : 'F U T, 0, 1, 0',
	X =  -279.868  mm,	Y =     0.000  mm,	Z =     0.000  mm,
	W =  -167.363 deg,	P =     0.003 deg,	R =   -75.545 deg
};
P[3094]{
   GP1:
	UF : 7, UT : 3,	CONFIG : 'F U T, 0, 1, 0',
	X =  -279.064  mm,	Y =    21.046  mm,	Z =     0.001  mm,
	W =  -167.360 deg,	P =     0.007 deg,	R =   -79.288 deg
};
P[3095]{
   GP1:
	UF : 7, UT : 3,	CONFIG : 'F U T, 0, 1, 0',
	X =  -276.988  mm,	Y =    39.955  mm,	Z =     0.001  mm,
	W =  -167.359 deg,	P =     0.011 deg,	R =   -83.162 deg
};
P[3096]{
   GP1:
	UF : 7, UT : 3,	CONFIG : 'F U T, 0, 0, 0',
	X =  -273.646  mm,	Y =    58.627  mm,	Z =     0.001  mm,
	W =  -167.358 deg,	P =     0.015 deg,	R =   -87.043 deg
};
P[3097]{
   GP1:
	UF : 7, UT : 3,	CONFIG : 'F U T, 0, 0, 0',
	X =  -269.041  mm,	Y =    77.049  mm,	Z =     0.004  mm,
	W =  -167.357 deg,	P =     0.019 deg,	R =   -90.920 deg
};
P[3098]{
   GP1:
	UF : 7, UT : 3,	CONFIG : 'F U T, 0, 0, 0',
	X =  -262.533  mm,	Y =    96.954  mm,	Z =     0.023  mm,
	W =  -167.440 deg,	P =     0.118 deg,	R =   -95.217 deg
};
P[3099]{
   GP1:
	UF : 7, UT : 3,	CONFIG : 'F U T, 0, 0, 0',
	X =  -255.965  mm,	Y =   113.152  mm,	Z =     0.061  mm,
	W =  -167.663 deg,	P =     0.216 deg,	R =   -98.794 deg
};
P[3100]{
   GP1:
	UF : 7, UT : 3,	CONFIG : 'F U T, 0, 0, 0',
	X =  -249.618  mm,	Y =   126.542  mm,	Z =     0.083  mm,
	W =  -167.798 deg,	P =     0.146 deg,	R =  -101.831 deg
};
P[3101]{
   GP1:
	UF : 7, UT : 3,	CONFIG : 'F U T, 0, 0, 0',
	X =  -242.109  mm,	Y =   140.359  mm,	Z =     0.075  mm,
	W =  -167.725 deg,	P =     0.010 deg,	R =  -105.057 deg
};
P[3102]{
   GP1:
	UF : 7, UT : 3,	CONFIG : 'F U T, 0, 0, 0',
	X =  -235.595  mm,	Y =   151.041  mm,	Z =     0.052  mm,
	W =  -167.563 deg,	P =    -0.042 deg,	R =  -107.619 deg
};
P[3103]{
   GP1:
	UF : 7, UT : 3,	CONFIG : 'F U T, 0, 0, 0',
	X =  -228.604  mm,	Y =   161.430  mm,	Z =     0.031  mm,
	W =  -167.398 deg,	P =    -0.079 deg,	R =  -110.179 deg
};
P[3104]{
   GP1:
	UF : 7, UT : 3,	CONFIG : 'F U T, 0, 0, 0',
	X =  -218.229  mm,	Y =   175.201  mm,	Z =     0.016  mm,
	W =  -167.302 deg,	P =    -0.029 deg,	R =  -113.700 deg
};
P[3105]{
   GP1:
	UF : 7, UT : 3,	CONFIG : 'F U T, 0, 0, 0',
	X =  -207.855  mm,	Y =   187.393  mm,	Z =     0.018  mm,
	W =  -167.353 deg,	P =     0.002 deg,	R =  -116.985 deg
};
P[3106]{
   GP1:
	UF : 7, UT : 3,	CONFIG : 'F U T, 0, 0, 0',
	X =  -196.771  mm,	Y =   199.003  mm,	Z =     0.024  mm,
	W =  -167.406 deg,	P =     0.027 deg,	R =  -120.261 deg
};
P[3107]{
   GP1:
	UF : 7, UT : 3,	CONFIG : 'F U T, 0, 0, 0',
	X =  -186.353  mm,	Y =   208.794  mm,	Z =     0.026  mm,
	W =  -167.412 deg,	P =     0.015 deg,	R =  -123.195 deg
};
P[3108]{
   GP1:
	UF : 7, UT : 3,	CONFIG : 'F U T, 0, 0, 0',
	X =  -175.444  mm,	Y =   218.034  mm,	Z =     0.024  mm,
	W =  -167.415 deg,	P =     0.003 deg,	R =  -126.129 deg
};
P[3109]{
   GP1:
	UF : 7, UT : 3,	CONFIG : 'F U T, 0, 0, 0',
	X =  -164.066  mm,	Y =   226.716  mm,	Z =     0.019  mm,
	W =  -167.418 deg,	P =    -0.010 deg,	R =  -129.059 deg
};
P[3110]{
   GP1:
	UF : 7, UT : 3,	CONFIG : 'F U T, 0, 0, 0',
	X =  -151.992  mm,	Y =   234.983  mm,	Z =     0.012  mm,
	W =  -167.402 deg,	P =    -0.010 deg,	R =  -132.049 deg
};
P[3111]{
   GP1:
	UF : 7, UT : 3,	CONFIG : 'F U T, 0, 0, 0',
	X =  -139.483  mm,	Y =   242.616  mm,	Z =     0.006  mm,
	W =  -167.386 deg,	P =    -0.009 deg,	R =  -135.034 deg
};
P[3112]{
   GP1:
	UF : 7, UT : 3,	CONFIG : 'F U T, 0, 0, 0',
	X =  -126.670  mm,	Y =   249.552  mm,	Z =     0.002  mm,
	W =  -167.370 deg,	P =    -0.007 deg,	R =  -138.036 deg
};
P[3113]{
   GP1:
	UF : 7, UT : 3,	CONFIG : 'F U T, 0, 0, 0',
	X =  -113.474  mm,	Y =   255.822  mm,	Z =     0.002  mm,
	W =  -167.355 deg,	P =    -0.002 deg,	R =  -141.030 deg
};
P[3114]{
   GP1:
	UF : 7, UT : 3,	CONFIG : 'F U T, 0, 0, 0',
	X =   -96.101  mm,	Y =   262.843  mm,	Z =     0.002  mm,
	W =  -167.356 deg,	P =    -0.001 deg,	R =  -144.856 deg
};
P[3115]{
   GP1:
	UF : 7, UT : 3,	CONFIG : 'F U T, 0, 0, 0',
	X =   -78.337  mm,	Y =   268.675  mm,	Z =     0.002  mm,
	W =  -167.357 deg,	P =    -0.001 deg,	R =  -148.691 deg
};
P[3116]{
   GP1:
	UF : 7, UT : 3,	CONFIG : 'F U T, 0, 0, 0',
	X =   -60.186  mm,	Y =   273.308  mm,	Z =     0.002  mm,
	W =  -167.358 deg,	P =     0.000 deg,	R =  -152.520 deg
};
P[3117]{
   GP1:
	UF : 7, UT : 3,	CONFIG : 'F U T, 0, 0, 0',
	X =   -41.782  mm,	Y =   276.717  mm,	Z =     0.002  mm,
	W =  -167.359 deg,	P =     0.000 deg,	R =  -156.351 deg
};
P[3118]{
   GP1:
	UF : 7, UT : 3,	CONFIG : 'F U T, 0, 0, 0',
	X =   -23.137  mm,	Y =   278.894  mm,	Z =     0.001  mm,
	W =  -167.360 deg,	P =     0.001 deg,	R =  -160.172 deg
};
P[3119]{
   GP1:
	UF : 7, UT : 3,	CONFIG : 'F U T, 0, 0, 0',
	X =    -4.451  mm,	Y =   279.818  mm,	Z =     0.000  mm,
	W =  -167.361 deg,	P =     0.001 deg,	R =  -164.006 deg
};
P[3120]{
   GP1:
	UF : 7, UT : 3,	CONFIG : 'F U T, 0, 0, 0',
	X =    14.224  mm,	Y =   279.494  mm,	Z =     0.001  mm,
	W =  -167.362 deg,	P =     0.001 deg,	R =  -167.847 deg
};
P[3121]{
   GP1:
	UF : 7, UT : 3,	CONFIG : 'F U T, 0, 0, 0',
	X =    32.830  mm,	Y =   277.926  mm,	Z =     0.001  mm,
	W =  -167.363 deg,	P =     0.001 deg,	R =  -171.688 deg
};
P[3122]{
   GP1:
	UF : 7, UT : 3,	CONFIG : 'F U T, 0, 0, 0',
	X =    52.590  mm,	Y =   274.869  mm,	Z =     0.001  mm,
	W =  -167.363 deg,	P =     0.001 deg,	R =  -175.784 deg
};
P[3123]{
   GP1:
	UF : 7, UT : 3,	CONFIG : 'F U T, 0, 0, 0',
	X =    72.085  mm,	Y =   270.414  mm,	Z =     0.001  mm,
	W =  -167.363 deg,	P =     0.000 deg,	R =  -179.879 deg
};
P[3124]{
   GP1:
	UF : 7, UT : 3,	CONFIG : 'F U T, 0, 0, 0',
	X =    91.218  mm,	Y =   264.579  mm,	Z =     0.001  mm,
	W =  -167.363 deg,	P =     0.000 deg,	R =   176.024 deg
};
P[3125]{
   GP1:
	UF : 7, UT : 3,	CONFIG : 'F U T, 0, 0, 0',
	X =   109.910  mm,	Y =   257.368  mm,	Z =     0.000  mm,
	W =  -167.363 deg,	P =     0.000 deg,	R =   171.935 deg
};
P[3126]{
   GP1:
	UF : 7, UT : 3,	CONFIG : 'F U T, 0, 0, 0',
	X =   127.991  mm,	Y =   248.870  mm,	Z =     0.000  mm,
	W =  -167.363 deg,	P =     0.000 deg,	R =   167.836 deg
};
P[3127]{
   GP1:
	UF : 7, UT : 3,	CONFIG : 'F U T, 0, 0, 0',
	X =   145.354  mm,	Y =   239.145  mm,	Z =     0.001  mm,
	W =  -167.363 deg,	P =     0.000 deg,	R =   163.721 deg
};
P[3128]{
   GP1:
	UF : 7, UT : 3,	CONFIG : 'F U T, 0, 0, 0',
	X =   162.123  mm,	Y =   228.111  mm,	Z =     0.002  mm,
	W =  -167.363 deg,	P =    -0.001 deg,	R =   159.639 deg
};
P[3129]{
   GP1:
	UF : 7, UT : 3,	CONFIG : 'F U T, 0, 0, 0',
	X =   178.031  mm,	Y =   215.925  mm,	Z =     0.002  mm,
	W =  -167.363 deg,	P =    -0.001 deg,	R =   155.551 deg
};
P[3130]{
   GP1:
	UF : 7, UT : 3,	CONFIG : 'F U T, 0, 0, 0',
	X =   193.021  mm,	Y =   202.631  mm,	Z =     0.001  mm,
	W =  -167.363 deg,	P =    -0.001 deg,	R =   151.462 deg
};
P[3131]{
   GP1:
	UF : 7, UT : 3,	CONFIG : 'F U T, 0, 0, 0',
	X =   206.971  mm,	Y =   188.362  mm,	Z =     0.001  mm,
	W =  -167.363 deg,	P =    -0.001 deg,	R =   147.356 deg
};
P[3132]{
   GP1:
	UF : 7, UT : 3,	CONFIG : 'F U T, 0, 0, 0',
	X =   220.182  mm,	Y =   172.743  mm,	Z =     0.000  mm,
	W =  -167.363 deg,	P =    -0.001 deg,	R =   143.177 deg
};
P[3133]{
   GP1:
	UF : 7, UT : 3,	CONFIG : 'F U T, 0, 0, 0',
	X =   232.201  mm,	Y =   156.211  mm,	Z =     0.001  mm,
	W =  -167.363 deg,	P =    -0.001 deg,	R =   138.993 deg
};
P[3134]{
   GP1:
	UF : 7, UT : 3,	CONFIG : 'F U T, 0, 0, 0',
	X =   242.979  mm,	Y =   138.854  mm,	Z =     0.001  mm,
	W =  -167.363 deg,	P =    -0.001 deg,	R =   134.808 deg
};
P[3135]{
   GP1:
	UF : 7, UT : 3,	CONFIG : 'F U T, 0, 0, 0',
	X =   252.460  mm,	Y =   120.778  mm,	Z =     0.001  mm,
	W =  -167.363 deg,	P =    -0.001 deg,	R =   130.618 deg
};
P[3136]{
   GP1:
	UF : 7, UT : 3,	CONFIG : 'F U T, 0, 0, 0',
	X =   260.598  mm,	Y =   102.046  mm,	Z =     0.001  mm,
	W =  -167.363 deg,	P =    -0.001 deg,	R =   126.431 deg
};
P[3137]{
   GP1:
	UF : 7, UT : 3,	CONFIG : 'F U T, 0, 0, 0',
	X =   267.347  mm,	Y =    82.726  mm,	Z =     0.000  mm,
	W =  -167.363 deg,	P =    -0.001 deg,	R =   122.251 deg
};
P[3138]{
   GP1:
	UF : 7, UT : 3,	CONFIG : 'F U T, 0, 0, 0',
	X =   272.657  mm,	Y =    63.055  mm,	Z =     0.000  mm,
	W =  -167.363 deg,	P =    -0.001 deg,	R =   118.055 deg
};
P[3139]{
   GP1:
	UF : 7, UT : 3,	CONFIG : 'F U T, 0, 0, 0',
	X =   276.544  mm,	Y =    42.917  mm,	Z =     0.000  mm,
	W =  -167.363 deg,	P =    -0.001 deg,	R =   113.886 deg
};
P[3140]{
   GP1:
	UF : 7, UT : 3,	CONFIG : 'F U T, 0, 0, 0',
	X =   278.932  mm,	Y =    22.664  mm,	Z =     0.000  mm,
	W =  -167.364 deg,	P =    -0.001 deg,	R =   109.693 deg
};
P[3141]{
   GP1:
	UF : 7, UT : 3,	CONFIG : 'F U T, 0, 0, 0',
	X =   279.868  mm,	Y =     0.000  mm,	Z =     0.000  mm,
	W =  -167.364 deg,	P =    -0.001 deg,	R =   105.656 deg
};
P[3142]{
   GP1:
	UF : 7, UT : 3,	CONFIG : 'F U T, 0, 0, 0',
	X =   279.868  mm,	Y =     0.000  mm,	Z =     0.000  mm,
	W =  -167.364 deg,	P =    -0.001 deg,	R =   105.656 deg
};
P[3143]{
   GP1:
	UF : 7, UT : 3,	CONFIG : 'F U T, 0, 0, 0',
	X =   279.868  mm,	Y =     0.000  mm,	Z =     0.000  mm,
	W =  -167.364 deg,	P =    -0.001 deg,	R =   105.656 deg
};
P[3144]{
   GP1:
	UF : 7, UT : 3,	CONFIG : 'F U T, 0, 0, 0',
	X =   279.868  mm,	Y =     0.000  mm,	Z =     0.000  mm,
	W =  -167.364 deg,	P =    -0.001 deg,	R =   105.656 deg
};
P[3145]{
   GP1:
	UF : 7, UT : 3,	CONFIG : 'F U T, 0, 0, 0',
	X =   276.733  mm,	Y =     0.000  mm,	Z =     0.000  mm,
	W =  -167.364 deg,	P =    -0.001 deg,	R =   105.609 deg
};
P[3146]{
   GP1:
	UF : 7, UT : 3,	CONFIG : 'F U T, 0, 0, 0',
	X =   276.733  mm,	Y =     0.000  mm,	Z =     0.000  mm,
	W =  -167.364 deg,	P =    -0.001 deg,	R =   105.609 deg
};
P[3147]{
   GP1:
	UF : 7, UT : 3,	CONFIG : 'F U T, 0, 0, 0',
	X =   276.733  mm,	Y =     0.000  mm,	Z =     0.000  mm,
	W =  -167.364 deg,	P =    -0.001 deg,	R =   105.609 deg
};
P[3148]{
   GP1:
	UF : 7, UT : 3,	CONFIG : 'F U T, 0, 0, 0',
	X =   276.733  mm,	Y =     0.000  mm,	Z =     0.000  mm,
	W =  -167.364 deg,	P =    -0.001 deg,	R =   105.609 deg
};
P[3149]{
   GP1:
	UF : 7, UT : 3,	CONFIG : 'F U T, 0, 0, 0',
	X =   275.905  mm,	Y =    21.226  mm,	Z =     0.000  mm,
	W =  -167.364 deg,	P =    -0.001 deg,	R =   109.460 deg
};
P[3150]{
   GP1:
	UF : 7, UT : 3,	CONFIG : 'F U T, 0, 0, 0',
	X =   273.728  mm,	Y =    40.594  mm,	Z =     0.000  mm,
	W =  -167.364 deg,	P =    -0.001 deg,	R =   113.496 deg
};
P[3151]{
   GP1:
	UF : 7, UT : 3,	CONFIG : 'F U T, 0, 0, 0',
	X =   270.194  mm,	Y =    59.777  mm,	Z =     0.000  mm,
	W =  -167.364 deg,	P =    -0.001 deg,	R =   117.530 deg
};
P[3152]{
   GP1:
	UF : 7, UT : 3,	CONFIG : 'F U T, 0, 0, 0',
	X =   265.315  mm,	Y =    78.661  mm,	Z =     0.000  mm,
	W =  -167.364 deg,	P =    -0.001 deg,	R =   121.564 deg
};
P[3153]{
   GP1:
	UF : 7, UT : 3,	CONFIG : 'F U T, 0, 0, 0',
	X =   259.109  mm,	Y =    97.152  mm,	Z =     0.001  mm,
	W =  -167.364 deg,	P =    -0.001 deg,	R =   125.598 deg
};
P[3154]{
   GP1:
	UF : 7, UT : 3,	CONFIG : 'F U T, 0, 0, 0',
	X =   251.620  mm,	Y =   115.156  mm,	Z =     0.001  mm,
	W =  -167.364 deg,	P =    -0.001 deg,	R =   129.634 deg
};
P[3155]{
   GP1:
	UF : 7, UT : 3,	CONFIG : 'F U T, 0, 0, 0',
	X =   242.888  mm,	Y =   132.584  mm,	Z =     0.001  mm,
	W =  -167.364 deg,	P =    -0.001 deg,	R =   133.669 deg
};
P[3156]{
   GP1:
	UF : 7, UT : 3,	CONFIG : 'F U T, 0, 0, 0',
	X =   232.967  mm,	Y =   149.333  mm,	Z =     0.001  mm,
	W =  -167.364 deg,	P =     0.000 deg,	R =   137.709 deg
};
P[3157]{
   GP1:
	UF : 7, UT : 3,	CONFIG : 'F U T, 0, 0, 0',
	X =   221.870  mm,	Y =   165.371  mm,	Z =     0.000  mm,
	W =  -167.364 deg,	P =     0.000 deg,	R =   141.745 deg
};
P[3158]{
   GP1:
	UF : 7, UT : 3,	CONFIG : 'F U T, 0, 0, 0',
	X =   209.680  mm,	Y =   180.580  mm,	Z =     0.000  mm,
	W =  -167.364 deg,	P =    -0.001 deg,	R =   145.782 deg
};
P[3159]{
   GP1:
	UF : 7, UT : 3,	CONFIG : 'F U T, 0, 0, 0',
	X =   197.868  mm,	Y =   193.462  mm,	Z =     0.001  mm,
	W =  -167.364 deg,	P =    -0.001 deg,	R =   149.408 deg
};
P[3160]{
   GP1:
	UF : 7, UT : 3,	CONFIG : 'F U T, 0, 0, 0',
	X =   185.246  mm,	Y =   205.569  mm,	Z =     0.001  mm,
	W =  -167.364 deg,	P =    -0.001 deg,	R =   153.036 deg
};
P[3161]{
   GP1:
	UF : 7, UT : 3,	CONFIG : 'F U T, 0, 0, 0',
	X =   171.859  mm,	Y =   216.886  mm,	Z =     0.001  mm,
	W =  -167.365 deg,	P =    -0.001 deg,	R =   156.653 deg
};
P[3162]{
   GP1:
	UF : 7, UT : 3,	CONFIG : 'F U T, 0, 0, 0',
	X =   157.807  mm,	Y =   227.317  mm,	Z =     0.001  mm,
	W =  -167.365 deg,	P =    -0.001 deg,	R =   160.279 deg
};
P[3163]{
   GP1:
	UF : 7, UT : 3,	CONFIG : 'F U T, 0, 0, 0',
	X =   143.054  mm,	Y =   236.871  mm,	Z =     0.001  mm,
	W =  -167.365 deg,	P =     0.000 deg,	R =   163.888 deg
};
P[3164]{
   GP1:
	UF : 7, UT : 3,	CONFIG : 'F U T, 0, 0, 0',
	X =   127.887  mm,	Y =   245.400  mm,	Z =     0.001  mm,
	W =  -167.365 deg,	P =     0.000 deg,	R =   167.530 deg
};
P[3165]{
   GP1:
	UF : 7, UT : 3,	CONFIG : 'F U T, 0, 0, 0',
	X =   112.109  mm,	Y =   252.995  mm,	Z =     0.001  mm,
	W =  -167.366 deg,	P =     0.000 deg,	R =   171.150 deg
};
P[3166]{
   GP1:
	UF : 7, UT : 3,	CONFIG : 'F U T, 0, 0, 0',
	X =    95.953  mm,	Y =   259.557  mm,	Z =     0.001  mm,
	W =  -167.366 deg,	P =     0.000 deg,	R =   174.785 deg
};
P[3167]{
   GP1:
	UF : 7, UT : 3,	CONFIG : 'F U T, 0, 0, 0',
	X =    79.292  mm,	Y =   265.125  mm,	Z =     0.001  mm,
	W =  -167.366 deg,	P =     0.000 deg,	R =   178.394 deg
};
P[3168]{
   GP1:
	UF : 7, UT : 3,	CONFIG : 'F U T, 0, 0, 0',
	X =    62.392  mm,	Y =   269.594  mm,	Z =     0.001  mm,
	W =  -167.367 deg,	P =     0.001 deg,	R =  -177.982 deg
};
P[3169]{
   GP1:
	UF : 7, UT : 3,	CONFIG : 'F U T, 0, 0, 0',
	X =    42.642  mm,	Y =   273.415  mm,	Z =     0.001  mm,
	W =  -167.367 deg,	P =     0.001 deg,	R =  -173.812 deg
};
P[3170]{
   GP1:
	UF : 7, UT : 3,	CONFIG : 'F U T, 0, 0, 0',
	X =    22.592  mm,	Y =   275.794  mm,	Z =     0.001  mm,
	W =  -167.366 deg,	P =     0.001 deg,	R =  -169.659 deg
};
P[3171]{
   GP1:
	UF : 7, UT : 3,	CONFIG : 'F U T, 0, 0, 0',
	X =     2.512  mm,	Y =   276.707  mm,	Z =     0.001  mm,
	W =  -167.366 deg,	P =     0.001 deg,	R =  -165.486 deg
};
P[3172]{
   GP1:
	UF : 7, UT : 3,	CONFIG : 'F U T, 0, 0, 0',
	X =   -17.558  mm,	Y =   276.164  mm,	Z =     0.001  mm,
	W =  -167.366 deg,	P =     0.001 deg,	R =  -161.308 deg
};
P[3173]{
   GP1:
	UF : 7, UT : 3,	CONFIG : 'F U T, 0, 0, 0',
	X =   -37.613  mm,	Y =   274.151  mm,	Z =     0.001  mm,
	W =  -167.366 deg,	P =     0.001 deg,	R =  -157.147 deg
};
P[3174]{
   GP1:
	UF : 7, UT : 3,	CONFIG : 'F U T, 0, 0, 0',
	X =   -57.429  mm,	Y =   270.692  mm,	Z =     0.002  mm,
	W =  -167.366 deg,	P =     0.001 deg,	R =  -152.980 deg
};
P[3175]{
   GP1:
	UF : 7, UT : 3,	CONFIG : 'F U T, 0, 0, 0',
	X =   -76.878  mm,	Y =   265.826  mm,	Z =     0.002  mm,
	W =  -167.366 deg,	P =     0.001 deg,	R =  -148.798 deg
};
P[3176]{
   GP1:
	UF : 7, UT : 3,	CONFIG : 'F U T, 0, 0, 0',
	X =   -96.036  mm,	Y =   259.522  mm,	Z =     0.002  mm,
	W =  -167.366 deg,	P =     0.001 deg,	R =  -144.641 deg
};
P[3177]{
   GP1:
	UF : 7, UT : 3,	CONFIG : 'F U T, 0, 0, 0',
	X =  -111.566  mm,	Y =   253.237  mm,	Z =     0.002  mm,
	W =  -167.372 deg,	P =    -0.004 deg,	R =  -141.162 deg
};
P[3178]{
   GP1:
	UF : 7, UT : 3,	CONFIG : 'F U T, 0, 0, 0',
	X =  -126.717  mm,	Y =   245.999  mm,	Z =     0.003  mm,
	W =  -167.378 deg,	P =    -0.009 deg,	R =  -137.691 deg
};
P[3179]{
   GP1:
	UF : 7, UT : 3,	CONFIG : 'F U T, 0, 0, 0',
	X =  -141.414  mm,	Y =   237.862  mm,	Z =     0.007  mm,
	W =  -167.384 deg,	P =    -0.013 deg,	R =  -134.223 deg
};
P[3180]{
   GP1:
	UF : 7, UT : 3,	CONFIG : 'F U T, 0, 0, 0',
	X =  -156.114  mm,	Y =   228.483  mm,	Z =     0.013  mm,
	W =  -167.412 deg,	P =    -0.004 deg,	R =  -130.609 deg
};
P[3181]{
   GP1:
	UF : 7, UT : 3,	CONFIG : 'F U T, 0, 0, 0',
	X =  -170.188  mm,	Y =   218.199  mm,	Z =     0.018  mm,
	W =  -167.439 deg,	P =     0.009 deg,	R =  -126.993 deg
};
P[3182]{
   GP1:
	UF : 7, UT : 3,	CONFIG : 'F U T, 0, 0, 0',
	X =  -183.602  mm,	Y =   207.045  mm,	Z =     0.021  mm,
	W =  -167.465 deg,	P =     0.025 deg,	R =  -123.382 deg
};
P[3183]{
   GP1:
	UF : 7, UT : 3,	CONFIG : 'F U T, 0, 0, 0',
	X =  -193.273  mm,	Y =   198.054  mm,	Z =     0.021  mm,
	W =  -167.437 deg,	P =     0.022 deg,	R =  -120.647 deg
};
P[3184]{
   GP1:
	UF : 7, UT : 3,	CONFIG : 'F U T, 0, 0, 0',
	X =  -202.505  mm,	Y =   188.601  mm,	Z =     0.019  mm,
	W =  -167.411 deg,	P =     0.016 deg,	R =  -117.915 deg
};
P[3185]{
   GP1:
	UF : 7, UT : 3,	CONFIG : 'F U T, 0, 0, 0',
	X =  -211.271  mm,	Y =   178.719  mm,	Z =     0.017  mm,
	W =  -167.385 deg,	P =     0.008 deg,	R =  -115.181 deg
};
P[3186]{
   GP1:
	UF : 7, UT : 3,	CONFIG : 'F U T, 0, 0, 0',
	X =  -223.630  mm,	Y =   162.985  mm,	Z =     0.024  mm,
	W =  -167.440 deg,	P =    -0.026 deg,	R =  -111.038 deg
};
P[3187]{
   GP1:
	UF : 7, UT : 3,	CONFIG : 'F U T, 0, 0, 0',
	X =  -231.027  mm,	Y =   152.320  mm,	Z =     0.037  mm,
	W =  -167.573 deg,	P =    -0.004 deg,	R =  -108.342 deg
};
P[3188]{
   GP1:
	UF : 7, UT : 3,	CONFIG : 'F U T, 0, 0, 0',
	X =  -237.909  mm,	Y =   141.334  mm,	Z =     0.052  mm,
	W =  -167.705 deg,	P =     0.030 deg,	R =  -105.642 deg
};
P[3189]{
   GP1:
	UF : 7, UT : 3,	CONFIG : 'F U T, 0, 0, 0',
	X =  -245.856  mm,	Y =   126.999  mm,	Z =     0.059  mm,
	W =  -167.782 deg,	P =     0.125 deg,	R =  -102.253 deg
};
P[3190]{
   GP1:
	UF : 7, UT : 3,	CONFIG : 'F U T, 0, 0, 0',
	X =  -252.468  mm,	Y =   113.288  mm,	Z =     0.045  mm,
	W =  -167.670 deg,	P =     0.172 deg,	R =   -99.108 deg
};
P[3191]{
   GP1:
	UF : 7, UT : 3,	CONFIG : 'F U T, 0, 0, 0',
	X =  -259.258  mm,	Y =    96.750  mm,	Z =     0.018  mm,
	W =  -167.464 deg,	P =     0.095 deg,	R =   -95.403 deg
};
P[3192]{
   GP1:
	UF : 7, UT : 3,	CONFIG : 'F U T, 0, 0, 0',
	X =  -262.824  mm,	Y =    86.595  mm,	Z =     0.008  mm,
	W =  -167.415 deg,	P =     0.058 deg,	R =   -93.198 deg
};
P[3193]{
   GP1:
	UF : 7, UT : 3,	CONFIG : 'F U T, 0, 0, 0',
	X =  -265.968  mm,	Y =    76.377  mm,	Z =     0.004  mm,
	W =  -167.370 deg,	P =     0.018 deg,	R =   -90.979 deg
};
P[3194]{
   GP1:
	UF : 7, UT : 3,	CONFIG : 'F U T, 0, 0, 0',
	X =  -270.541  mm,	Y =    58.149  mm,	Z =     0.001  mm,
	W =  -167.367 deg,	P =     0.014 deg,	R =   -87.066 deg
};
P[3195]{
   GP1:
	UF : 7, UT : 3,	CONFIG : 'F U T, 0, 1, 0',
	X =  -273.877  mm,	Y =    39.572  mm,	Z =     0.001  mm,
	W =  -167.365 deg,	P =     0.011 deg,	R =   -83.168 deg
};
P[3196]{
   GP1:
	UF : 7, UT : 3,	CONFIG : 'F U T, 0, 1, 0',
	X =  -275.941  mm,	Y =    20.790  mm,	Z =     0.001  mm,
	W =  -167.364 deg,	P =     0.007 deg,	R =   -79.274 deg
};
P[3197]{
   GP1:
	UF : 7, UT : 3,	CONFIG : 'F U T, 0, 1, 0',
	X =  -276.733  mm,	Y =     0.000  mm,	Z =     0.000  mm,
	W =  -167.363 deg,	P =     0.002 deg,	R =   -75.530 deg
};
P[3198]{
   GP1:
	UF : 7, UT : 3,	CONFIG : 'F U T, 0, 1, 0',
	X =  -276.733  mm,	Y =     0.000  mm,	Z =     0.000  mm,
	W =  -167.363 deg,	P =     0.002 deg,	R =   -75.530 deg
};
P[3199]{
   GP1:
	UF : 7, UT : 3,	CONFIG : 'F U T, 0, 1, 0',
	X =  -276.733  mm,	Y =     0.000  mm,	Z =     0.000  mm,
	W =  -167.363 deg,	P =     0.002 deg,	R =   -75.530 deg
};
P[3200]{
   GP1:
	UF : 7, UT : 3,	CONFIG : 'F U T, 0, 1, 0',
	X =  -276.733  mm,	Y =     0.000  mm,	Z =     0.000  mm,
	W =  -167.363 deg,	P =     0.002 deg,	R =   -75.530 deg
};
P[3201]{
   GP1:
	UF : 7, UT : 3,	CONFIG : 'F U T, 0, 1, 0',
	X =  -273.599  mm,	Y =     0.000  mm,	Z =     0.000  mm,
	W =  -167.363 deg,	P =     0.001 deg,	R =   -75.500 deg
};
P[3202]{
   GP1:
	UF : 7, UT : 3,	CONFIG : 'F U T, 0, 1, 0',
	X =  -273.599  mm,	Y =     0.000  mm,	Z =     0.000  mm,
	W =  -167.363 deg,	P =     0.001 deg,	R =   -75.500 deg
};
P[3203]{
   GP1:
	UF : 7, UT : 3,	CONFIG : 'F U T, 0, 1, 0',
	X =  -273.599  mm,	Y =     0.000  mm,	Z =     0.000  mm,
	W =  -167.363 deg,	P =     0.001 deg,	R =   -75.500 deg
};
P[3204]{
   GP1:
	UF : 7, UT : 3,	CONFIG : 'F U T, 0, 1, 0',
	X =  -273.599  mm,	Y =     0.000  mm,	Z =     0.000  mm,
	W =  -167.363 deg,	P =     0.001 deg,	R =   -75.500 deg
};
P[3205]{
   GP1:
	UF : 7, UT : 3,	CONFIG : 'F U T, 0, 1, 0',
	X =  -272.794  mm,	Y =    20.828  mm,	Z =     0.000  mm,
	W =  -167.368 deg,	P =     0.007 deg,	R =   -79.328 deg
};
P[3206]{
   GP1:
	UF : 7, UT : 3,	CONFIG : 'F U T, 0, 1, 0',
	X =  -270.664  mm,	Y =    39.897  mm,	Z =     0.001  mm,
	W =  -167.373 deg,	P =     0.011 deg,	R =   -83.333 deg
};
P[3207]{
   GP1:
	UF : 7, UT : 3,	CONFIG : 'F U T, 0, 0, 0',
	X =  -267.205  mm,	Y =    58.768  mm,	Z =     0.001  mm,
	W =  -167.379 deg,	P =     0.015 deg,	R =   -87.337 deg
};
P[3208]{
   GP1:
	UF : 7, UT : 3,	CONFIG : 'F U T, 0, 0, 0',
	X =  -262.446  mm,	Y =    77.283  mm,	Z =     0.003  mm,
	W =  -167.385 deg,	P =     0.018 deg,	R =   -91.355 deg
};
P[3209]{
   GP1:
	UF : 7, UT : 3,	CONFIG : 'F U T, 0, 0, 0',
	X =  -259.059  mm,	Y =    87.969  mm,	Z =     0.007  mm,
	W =  -167.443 deg,	P =     0.051 deg,	R =   -93.716 deg
};
P[3210]{
   GP1:
	UF : 7, UT : 3,	CONFIG : 'F U T, 0, 0, 0',
	X =  -255.209  mm,	Y =    98.594  mm,	Z =     0.014  mm,
	W =  -167.503 deg,	P =     0.081 deg,	R =   -96.059 deg
};
P[3211]{
   GP1:
	UF : 7, UT : 3,	CONFIG : 'F U T, 0, 0, 0',
	X =  -247.388  mm,	Y =   116.851  mm,	Z =     0.031  mm,
	W =  -167.711 deg,	P =     0.136 deg,	R =  -100.229 deg
};
P[3212]{
   GP1:
	UF : 7, UT : 3,	CONFIG : 'F U T, 0, 0, 0',
	X =  -240.310  mm,	Y =   130.767  mm,	Z =     0.036  mm,
	W =  -167.765 deg,	P =     0.103 deg,	R =  -103.525 deg
};
P[3213]{
   GP1:
	UF : 7, UT : 3,	CONFIG : 'F U T, 0, 0, 0',
	X =  -229.808  mm,	Y =   148.452  mm,	Z =     0.026  mm,
	W =  -167.630 deg,	P =     0.033 deg,	R =  -107.810 deg
};
P[3214]{
   GP1:
	UF : 7, UT : 3,	CONFIG : 'F U T, 0, 0, 0',
	X =  -222.648  mm,	Y =   158.995  mm,	Z =     0.019  mm,
	W =  -167.549 deg,	P =     0.020 deg,	R =  -110.477 deg
};
P[3215]{
   GP1:
	UF : 7, UT : 3,	CONFIG : 'F U T, 0, 0, 0',
	X =  -215.016  mm,	Y =   169.181  mm,	Z =     0.015  mm,
	W =  -167.467 deg,	P =     0.014 deg,	R =  -113.147 deg
};
P[3216]{
   GP1:
	UF : 7, UT : 3,	CONFIG : 'F U T, 0, 0, 0',
	X =  -203.565  mm,	Y =   182.792  mm,	Z =     0.014  mm,
	W =  -167.476 deg,	P =     0.025 deg,	R =  -116.864 deg
};
P[3217]{
   GP1:
	UF : 7, UT : 3,	CONFIG : 'F U T, 0, 0, 0',
	X =  -191.287  mm,	Y =   195.600  mm,	Z =     0.014  mm,
	W =  -167.487 deg,	P =     0.035 deg,	R =  -120.591 deg
};
P[3218]{
   GP1:
	UF : 7, UT : 3,	CONFIG : 'F U T, 0, 0, 0',
	X =  -179.210  mm,	Y =   206.726  mm,	Z =     0.014  mm,
	W =  -167.473 deg,	P =     0.024 deg,	R =  -124.015 deg
};
P[3219]{
   GP1:
	UF : 7, UT : 3,	CONFIG : 'F U T, 0, 0, 0',
	X =  -166.580  mm,	Y =   217.024  mm,	Z =     0.012  mm,
	W =  -167.459 deg,	P =     0.015 deg,	R =  -127.466 deg
};
P[3220]{
   GP1:
	UF : 7, UT : 3,	CONFIG : 'F U T, 0, 0, 0',
	X =  -153.220  mm,	Y =   226.661  mm,	Z =     0.009  mm,
	W =  -167.444 deg,	P =     0.008 deg,	R =  -130.880 deg
};
P[3221]{
   GP1:
	UF : 7, UT : 3,	CONFIG : 'F U T, 0, 0, 0',
	X =  -139.443  mm,	Y =   235.385  mm,	Z =     0.005  mm,
	W =  -167.426 deg,	P =     0.004 deg,	R =  -134.320 deg
};
P[3222]{
   GP1:
	UF : 7, UT : 3,	CONFIG : 'F U T, 0, 0, 0',
	X =  -125.034  mm,	Y =   243.342  mm,	Z =     0.003  mm,
	W =  -167.408 deg,	P =     0.001 deg,	R =  -137.729 deg
};
P[3223]{
   GP1:
	UF : 7, UT : 3,	CONFIG : 'F U T, 0, 0, 0',
	X =  -110.319  mm,	Y =   250.365  mm,	Z =     0.002  mm,
	W =  -167.390 deg,	P =     0.001 deg,	R =  -141.169 deg
};
P[3224]{
   GP1:
	UF : 7, UT : 3,	CONFIG : 'F U T, 0, 0, 0',
	X =   -95.166  mm,	Y =   256.501  mm,	Z =     0.002  mm,
	W =  -167.373 deg,	P =     0.003 deg,	R =  -144.602 deg
};
P[3225]{
   GP1:
	UF : 7, UT : 3,	CONFIG : 'F U T, 0, 0, 0',
	X =   -77.332  mm,	Y =   262.431  mm,	Z =     0.002  mm,
	W =  -167.372 deg,	P =     0.002 deg,	R =  -148.525 deg
};
P[3226]{
   GP1:
	UF : 7, UT : 3,	CONFIG : 'F U T, 0, 0, 0',
	X =   -59.177  mm,	Y =   267.115  mm,	Z =     0.002  mm,
	W =  -167.372 deg,	P =     0.002 deg,	R =  -152.456 deg
};
P[3227]{
   GP1:
	UF : 7, UT : 3,	CONFIG : 'F U T, 0, 0, 0',
	X =   -40.713  mm,	Y =   270.544  mm,	Z =     0.001  mm,
	W =  -167.371 deg,	P =     0.002 deg,	R =  -156.386 deg
};
P[3228]{
   GP1:
	UF : 7, UT : 3,	CONFIG : 'F U T, 0, 0, 0',
	X =   -22.038  mm,	Y =   272.696  mm,	Z =     0.001  mm,
	W =  -167.371 deg,	P =     0.002 deg,	R =  -160.308 deg
};
P[3229]{
   GP1:
	UF : 7, UT : 3,	CONFIG : 'F U T, 0, 0, 0',
	X =    -3.193  mm,	Y =   273.564  mm,	Z =     0.001  mm,
	W =  -167.371 deg,	P =     0.001 deg,	R =  -164.216 deg
};
P[3230]{
   GP1:
	UF : 7, UT : 3,	CONFIG : 'F U T, 0, 0, 0',
	X =    15.399  mm,	Y =   273.150  mm,	Z =     0.001  mm,
	W =  -167.370 deg,	P =     0.001 deg,	R =  -168.180 deg
};
P[3231]{
   GP1:
	UF : 7, UT : 3,	CONFIG : 'F U T, 0, 0, 0',
	X =    34.083  mm,	Y =   271.456  mm,	Z =     0.001  mm,
	W =  -167.370 deg,	P =     0.001 deg,	R =  -172.110 deg
};
P[3232]{
   GP1:
	UF : 7, UT : 3,	CONFIG : 'F U T, 0, 0, 0',
	X =    52.623  mm,	Y =   268.482  mm,	Z =     0.001  mm,
	W =  -167.369 deg,	P =     0.002 deg,	R =  -176.036 deg
};
P[3233]{
   GP1:
	UF : 7, UT : 3,	CONFIG : 'F U T, 0, 0, 0',
	X =    70.065  mm,	Y =   264.461  mm,	Z =     0.001  mm,
	W =  -167.369 deg,	P =     0.001 deg,	R =  -179.770 deg
};
P[3234]{
   GP1:
	UF : 7, UT : 3,	CONFIG : 'F U T, 0, 0, 0',
	X =    87.066  mm,	Y =   259.363  mm,	Z =     0.001  mm,
	W =  -167.369 deg,	P =     0.001 deg,	R =   176.463 deg
};
P[3235]{
   GP1:
	UF : 7, UT : 3,	CONFIG : 'F U T, 0, 0, 0',
	X =   103.873  mm,	Y =   253.101  mm,	Z =     0.000  mm,
	W =  -167.368 deg,	P =     0.001 deg,	R =   172.733 deg
};
P[3236]{
   GP1:
	UF : 7, UT : 3,	CONFIG : 'F U T, 0, 0, 0',
	X =   120.202  mm,	Y =   245.762  mm,	Z =     0.001  mm,
	W =  -167.368 deg,	P =     0.000 deg,	R =   168.999 deg
};
P[3237]{
   GP1:
	UF : 7, UT : 3,	CONFIG : 'F U T, 0, 0, 0',
	X =   135.948  mm,	Y =   237.419  mm,	Z =     0.001  mm,
	W =  -167.368 deg,	P =     0.000 deg,	R =   165.248 deg
};
P[3238]{
   GP1:
	UF : 7, UT : 3,	CONFIG : 'F U T, 0, 0, 0',
	X =   151.230  mm,	Y =   227.989  mm,	Z =     0.001  mm,
	W =  -167.367 deg,	P =     0.000 deg,	R =   161.522 deg
};
P[3239]{
   GP1:
	UF : 7, UT : 3,	CONFIG : 'F U T, 0, 0, 0',
	X =   165.803  mm,	Y =   217.616  mm,	Z =     0.001  mm,
	W =  -167.367 deg,	P =     0.000 deg,	R =   157.784 deg
};
P[3240]{
   GP1:
	UF : 7, UT : 3,	CONFIG : 'F U T, 0, 0, 0',
	X =   179.572  mm,	Y =   206.409  mm,	Z =     0.001  mm,
	W =  -167.367 deg,	P =     0.000 deg,	R =   154.015 deg
};
P[3241]{
   GP1:
	UF : 7, UT : 3,	CONFIG : 'F U T, 0, 0, 0',
	X =   192.714  mm,	Y =   194.192  mm,	Z =     0.001  mm,
	W =  -167.366 deg,	P =     0.000 deg,	R =   150.287 deg
};
P[3242]{
   GP1:
	UF : 7, UT : 3,	CONFIG : 'F U T, 0, 0, 0',
	X =   204.984  mm,	Y =   181.191  mm,	Z =     0.000  mm,
	W =  -167.366 deg,	P =     0.000 deg,	R =   146.546 deg
};
P[3243]{
   GP1:
	UF : 7, UT : 3,	CONFIG : 'F U T, 0, 0, 0',
	X =   217.387  mm,	Y =   166.105  mm,	Z =     0.000  mm,
	W =  -167.366 deg,	P =     0.000 deg,	R =   142.409 deg
};
P[3244]{
   GP1:
	UF : 7, UT : 3,	CONFIG : 'F U T, 0, 0, 0',
	X =   228.772  mm,	Y =   150.044  mm,	Z =     0.001  mm,
	W =  -167.365 deg,	P =     0.000 deg,	R =   138.303 deg
};
P[3245]{
   GP1:
	UF : 7, UT : 3,	CONFIG : 'F U T, 0, 0, 0',
	X =   238.960  mm,	Y =   133.231  mm,	Z =     0.001  mm,
	W =  -167.365 deg,	P =     0.000 deg,	R =   134.191 deg
};
P[3246]{
   GP1:
	UF : 7, UT : 3,	CONFIG : 'F U T, 0, 0, 0',
	X =   247.908  mm,	Y =   115.727  mm,	Z =     0.001  mm,
	W =  -167.365 deg,	P =     0.000 deg,	R =   130.081 deg
};
P[3247]{
   GP1:
	UF : 7, UT : 3,	CONFIG : 'F U T, 0, 0, 0',
	X =   255.560  mm,	Y =    97.666  mm,	Z =     0.000  mm,
	W =  -167.365 deg,	P =    -0.001 deg,	R =   125.962 deg
};
P[3248]{
   GP1:
	UF : 7, UT : 3,	CONFIG : 'F U T, 0, 0, 0',
	X =   261.917  mm,	Y =    79.069  mm,	Z =     0.000  mm,
	W =  -167.365 deg,	P =    -0.001 deg,	R =   121.848 deg
};
P[3249]{
   GP1:
	UF : 7, UT : 3,	CONFIG : 'F U T, 0, 0, 0',
	X =   266.922  mm,	Y =    60.067  mm,	Z =     0.000  mm,
	W =  -167.364 deg,	P =    -0.001 deg,	R =   117.736 deg
};
P[3250]{
   GP1:
	UF : 7, UT : 3,	CONFIG : 'F U T, 0, 0, 0',
	X =   270.540  mm,	Y =    40.737  mm,	Z =     0.000  mm,
	W =  -167.364 deg,	P =    -0.001 deg,	R =   113.626 deg
};
P[3251]{
   GP1:
	UF : 7, UT : 3,	CONFIG : 'F U T, 0, 0, 0',
	X =   272.767  mm,	Y =    21.173  mm,	Z =     0.000  mm,
	W =  -167.364 deg,	P =    -0.001 deg,	R =   109.520 deg
};
P[3252]{
   GP1:
	UF : 7, UT : 3,	CONFIG : 'F U T, 0, 0, 0',
	X =   273.599  mm,	Y =     0.000  mm,	Z =     0.000  mm,
	W =  -167.364 deg,	P =     0.000 deg,	R =   105.589 deg
};
P[3253]{
   GP1:
	UF : 7, UT : 3,	CONFIG : 'F U T, 0, 0, 0',
	X =   273.599  mm,	Y =     0.000  mm,	Z =     0.000  mm,
	W =  -167.364 deg,	P =     0.000 deg,	R =   105.589 deg
};
P[3254]{
   GP1:
	UF : 7, UT : 3,	CONFIG : 'F U T, 0, 0, 0',
	X =   273.599  mm,	Y =     0.000  mm,	Z =     0.000  mm,
	W =  -167.364 deg,	P =     0.000 deg,	R =   105.589 deg
};
P[3255]{
   GP1:
	UF : 7, UT : 3,	CONFIG : 'F U T, 0, 0, 0',
	X =   273.599  mm,	Y =     0.000  mm,	Z =     0.000  mm,
	W =  -167.364 deg,	P =     0.000 deg,	R =   105.589 deg
};
P[3256]{
   GP1:
	UF : 7, UT : 3,	CONFIG : 'F U T, 0, 0, 0',
	X =   270.465  mm,	Y =     0.000  mm,	Z =     0.000  mm,
	W =  -167.364 deg,	P =     0.000 deg,	R =   105.610 deg
};
P[3257]{
   GP1:
	UF : 7, UT : 3,	CONFIG : 'F U T, 0, 0, 0',
	X =   270.465  mm,	Y =     0.000  mm,	Z =     0.000  mm,
	W =  -167.364 deg,	P =     0.000 deg,	R =   105.610 deg
};
P[3258]{
   GP1:
	UF : 7, UT : 3,	CONFIG : 'F U T, 0, 0, 0',
	X =   270.465  mm,	Y =     0.000  mm,	Z =     0.000  mm,
	W =  -167.364 deg,	P =     0.000 deg,	R =   105.610 deg
};
P[3259]{
   GP1:
	UF : 7, UT : 3,	CONFIG : 'F U T, 0, 0, 0',
	X =   270.465  mm,	Y =     0.000  mm,	Z =     0.000  mm,
	W =  -167.364 deg,	P =     0.000 deg,	R =   105.610 deg
};
P[3260]{
   GP1:
	UF : 7, UT : 3,	CONFIG : 'F U T, 0, 0, 0',
	X =   269.541  mm,	Y =    22.179  mm,	Z =     0.000  mm,
	W =  -167.364 deg,	P =     0.000 deg,	R =   109.798 deg
};
P[3261]{
   GP1:
	UF : 7, UT : 3,	CONFIG : 'F U T, 0, 0, 0',
	X =   267.074  mm,	Y =    42.645  mm,	Z =     0.000  mm,
	W =  -167.365 deg,	P =    -0.001 deg,	R =   114.140 deg
};
P[3262]{
   GP1:
	UF : 7, UT : 3,	CONFIG : 'F U T, 0, 0, 0',
	X =   263.050  mm,	Y =    62.836  mm,	Z =     0.000  mm,
	W =  -167.365 deg,	P =    -0.001 deg,	R =   118.483 deg
};
P[3263]{
   GP1:
	UF : 7, UT : 3,	CONFIG : 'F U T, 0, 0, 0',
	X =   257.532  mm,	Y =    82.606  mm,	Z =     0.000  mm,
	W =  -167.366 deg,	P =    -0.001 deg,	R =   122.841 deg
};
P[3264]{
   GP1:
	UF : 7, UT : 3,	CONFIG : 'F U T, 0, 0, 0',
	X =   250.528  mm,	Y =   101.881  mm,	Z =     0.000  mm,
	W =  -167.367 deg,	P =    -0.001 deg,	R =   127.199 deg
};
P[3265]{
   GP1:
	UF : 7, UT : 3,	CONFIG : 'F U T, 0, 0, 0',
	X =   242.072  mm,	Y =   120.613  mm,	Z =     0.000  mm,
	W =  -167.367 deg,	P =     0.000 deg,	R =   131.551 deg
};
P[3266]{
   GP1:
	UF : 7, UT : 3,	CONFIG : 'F U T, 0, 0, 0',
	X =   232.211  mm,	Y =   138.647  mm,	Z =     0.000  mm,
	W =  -167.368 deg,	P =     0.000 deg,	R =   135.899 deg
};
P[3267]{
   GP1:
	UF : 7, UT : 3,	CONFIG : 'F U T, 0, 0, 0',
	X =   221.073  mm,	Y =   155.794  mm,	Z =     0.000  mm,
	W =  -167.369 deg,	P =     0.000 deg,	R =   140.272 deg
};
P[3268]{
   GP1:
	UF : 7, UT : 3,	CONFIG : 'F U T, 0, 0, 0',
	X =   208.504  mm,	Y =   172.254  mm,	Z =     0.000  mm,
	W =  -167.369 deg,	P =     0.001 deg,	R =   144.592 deg
};
P[3269]{
   GP1:
	UF : 7, UT : 3,	CONFIG : 'F U T, 0, 0, 0',
	X =   194.887  mm,	Y =   187.520  mm,	Z =     0.000  mm,
	W =  -167.370 deg,	P =     0.001 deg,	R =   148.967 deg
};
P[3270]{
   GP1:
	UF : 7, UT : 3,	CONFIG : 'F U T, 0, 0, 0',
	X =   182.780  mm,	Y =   199.336  mm,	Z =     0.000  mm,
	W =  -167.370 deg,	P =     0.001 deg,	R =   152.493 deg
};
P[3271]{
   GP1:
	UF : 7, UT : 3,	CONFIG : 'F U T, 0, 0, 0',
	X =   170.169  mm,	Y =   210.214  mm,	Z =     0.000  mm,
	W =  -167.370 deg,	P =     0.001 deg,	R =   156.074 deg
};
P[3272]{
   GP1:
	UF : 7, UT : 3,	CONFIG : 'F U T, 0, 0, 0',
	X =   156.769  mm,	Y =   220.381  mm,	Z =     0.000  mm,
	W =  -167.370 deg,	P =     0.001 deg,	R =   159.621 deg
};
P[3273]{
   GP1:
	UF : 7, UT : 3,	CONFIG : 'F U T, 0, 0, 0',
	X =   142.819  mm,	Y =   229.677  mm,	Z =     0.000  mm,
	W =  -167.371 deg,	P =     0.001 deg,	R =   163.181 deg
};
P[3274]{
   GP1:
	UF : 7, UT : 3,	CONFIG : 'F U T, 0, 0, 0',
	X =   128.331  mm,	Y =   238.063  mm,	Z =     0.000  mm,
	W =  -167.371 deg,	P =     0.001 deg,	R =   166.742 deg
};
P[3275]{
   GP1:
	UF : 7, UT : 3,	CONFIG : 'F U T, 0, 0, 0',
	X =   113.261  mm,	Y =   245.596  mm,	Z =     0.000  mm,
	W =  -167.372 deg,	P =     0.001 deg,	R =   170.283 deg
};
P[3276]{
   GP1:
	UF : 7, UT : 3,	CONFIG : 'F U T, 0, 0, 0',
	X =    97.796  mm,	Y =   252.151  mm,	Z =     0.000  mm,
	W =  -167.372 deg,	P =     0.002 deg,	R =   173.834 deg
};
P[3277]{
   GP1:
	UF : 7, UT : 3,	CONFIG : 'F U T, 0, 0, 0',
	X =    82.004  mm,	Y =   257.731  mm,	Z =     0.000  mm,
	W =  -167.372 deg,	P =     0.002 deg,	R =   177.394 deg
};
P[3278]{
   GP1:
	UF : 7, UT : 3,	CONFIG : 'F U T, 0, 0, 0',
	X =    65.894  mm,	Y =   262.305  mm,	Z =     0.000  mm,
	W =  -167.373 deg,	P =     0.002 deg,	R =  -179.039 deg
};
P[3279]{
   GP1:
	UF : 7, UT : 3,	CONFIG : 'F U T, 0, 0, 0',
	X =    49.508  mm,	Y =   265.883  mm,	Z =     0.000  mm,
	W =  -167.373 deg,	P =     0.003 deg,	R =  -175.483 deg
};
P[3280]{
   GP1:
	UF : 7, UT : 3,	CONFIG : 'F U T, 0, 0, 0',
	X =    31.091  mm,	Y =   268.658  mm,	Z =     0.000  mm,
	W =  -167.374 deg,	P =     0.002 deg,	R =  -171.534 deg
};
P[3281]{
   GP1:
	UF : 7, UT : 3,	CONFIG : 'F U T, 0, 0, 0',
	X =    12.506  mm,	Y =   270.169  mm,	Z =     0.000  mm,
	W =  -167.375 deg,	P =     0.002 deg,	R =  -167.587 deg
};
P[3282]{
   GP1:
	UF : 7, UT : 3,	CONFIG : 'F U T, 0, 0, 0',
	X =    -6.154  mm,	Y =   270.389  mm,	Z =     0.000  mm,
	W =  -167.376 deg,	P =     0.002 deg,	R =  -163.644 deg
};
P[3283]{
   GP1:
	UF : 7, UT : 3,	CONFIG : 'F U T, 0, 0, 0',
	X =   -24.761  mm,	Y =   269.316  mm,	Z =     0.000  mm,
	W =  -167.378 deg,	P =     0.002 deg,	R =  -159.696 deg
};
P[3284]{
   GP1:
	UF : 7, UT : 3,	CONFIG : 'F U T, 0, 0, 0',
	X =   -43.257  mm,	Y =   266.970  mm,	Z =     0.001  mm,
	W =  -167.379 deg,	P =     0.003 deg,	R =  -155.752 deg
};
P[3285]{
   GP1:
	UF : 7, UT : 3,	CONFIG : 'F U T, 0, 0, 0',
	X =   -61.499  mm,	Y =   263.371  mm,	Z =     0.001  mm,
	W =  -167.380 deg,	P =     0.003 deg,	R =  -151.798 deg
};
P[3286]{
   GP1:
	UF : 7, UT : 3,	CONFIG : 'F U T, 0, 0, 0',
	X =   -79.618  mm,	Y =   258.468  mm,	Z =     0.001  mm,
	W =  -167.381 deg,	P =     0.004 deg,	R =  -147.874 deg
};
P[3287]{
   GP1:
	UF : 7, UT : 3,	CONFIG : 'F U T, 0, 0, 0',
	X =   -97.038  mm,	Y =   252.440  mm,	Z =     0.001  mm,
	W =  -167.382 deg,	P =     0.005 deg,	R =  -143.885 deg
};
P[3288]{
   GP1:
	UF : 7, UT : 3,	CONFIG : 'F U T, 0, 0, 0',
	X =  -114.677  mm,	Y =   244.936  mm,	Z =     0.001  mm,
	W =  -167.408 deg,	P =     0.006 deg,	R =  -139.842 deg
};
P[3289]{
   GP1:
	UF : 7, UT : 3,	CONFIG : 'F U T, 0, 0, 0',
	X =  -131.731  mm,	Y =   236.210  mm,	Z =     0.002  mm,
	W =  -167.433 deg,	P =     0.011 deg,	R =  -135.796 deg
};
P[3290]{
   GP1:
	UF : 7, UT : 3,	CONFIG : 'F U T, 0, 0, 0',
	X =  -148.114  mm,	Y =   226.293  mm,	Z =     0.004  mm,
	W =  -167.458 deg,	P =     0.020 deg,	R =  -131.751 deg
};
P[3291]{
   GP1:
	UF : 7, UT : 3,	CONFIG : 'F U T, 0, 0, 0',
	X =  -163.472  mm,	Y =   215.453  mm,	Z =     0.005  mm,
	W =  -167.481 deg,	P =     0.025 deg,	R =  -127.777 deg
};
P[3292]{
   GP1:
	UF : 7, UT : 3,	CONFIG : 'F U T, 0, 0, 0',
	X =  -178.023  mm,	Y =   203.595  mm,	Z =     0.006  mm,
	W =  -167.504 deg,	P =     0.033 deg,	R =  -123.798 deg
};
P[3293]{
   GP1:
	UF : 7, UT : 3,	CONFIG : 'F U T, 0, 0, 0',
	X =  -191.688  mm,	Y =   190.790  mm,	Z =     0.006  mm,
	W =  -167.526 deg,	P =     0.044 deg,	R =  -119.808 deg
};
P[3294]{
   GP1:
	UF : 7, UT : 3,	CONFIG : 'F U T, 0, 0, 0',
	X =  -204.774  mm,	Y =   176.683  mm,	Z =     0.006  mm,
	W =  -167.541 deg,	P =     0.044 deg,	R =  -115.747 deg
};
P[3295]{
   GP1:
	UF : 7, UT : 3,	CONFIG : 'F U T, 0, 0, 0',
	X =  -216.777  mm,	Y =   161.719  mm,	Z =     0.008  mm,
	W =  -167.558 deg,	P =     0.045 deg,	R =  -111.674 deg
};
P[3296]{
   GP1:
	UF : 7, UT : 3,	CONFIG : 'F U T, 0, 0, 0',
	X =  -225.174  mm,	Y =   149.804  mm,	Z =     0.010  mm,
	W =  -167.643 deg,	P =     0.062 deg,	R =  -108.594 deg
};
P[3297]{
   GP1:
	UF : 7, UT : 3,	CONFIG : 'F U T, 0, 0, 0',
	X =  -232.907  mm,	Y =   137.493  mm,	Z =     0.013  mm,
	W =  -167.727 deg,	P =     0.088 deg,	R =  -105.506 deg
};
P[3298]{
   GP1:
	UF : 7, UT : 3,	CONFIG : 'F U T, 0, 0, 0',
	X =  -241.378  mm,	Y =   121.986  mm,	Z =     0.013  mm,
	W =  -167.738 deg,	P =     0.109 deg,	R =  -101.745 deg
};
P[3299]{
   GP1:
	UF : 7, UT : 3,	CONFIG : 'F U T, 0, 0, 0',
	X =  -246.047  mm,	Y =   112.277  mm,	Z =     0.010  mm,
	W =  -167.645 deg,	P =     0.094 deg,	R =   -99.466 deg
};
P[3300]{
   GP1:
	UF : 7, UT : 3,	CONFIG : 'F U T, 0, 0, 0',
	X =  -250.344  mm,	Y =   102.328  mm,	Z =     0.007  mm,
	W =  -167.553 deg,	P =     0.072 deg,	R =   -97.201 deg
};
P[3301]{
   GP1:
	UF : 7, UT : 3,	CONFIG : 'F U T, 0, 0, 0',
	X =  -254.770  mm,	Y =    90.746  mm,	Z =     0.004  mm,
	W =  -167.477 deg,	P =     0.047 deg,	R =   -94.570 deg
};
P[3302]{
   GP1:
	UF : 7, UT : 3,	CONFIG : 'F U T, 0, 0, 0',
	X =  -258.636  mm,	Y =    79.060  mm,	Z =     0.002  mm,
	W =  -167.404 deg,	P =     0.016 deg,	R =   -91.920 deg
};
P[3303]{
   GP1:
	UF : 7, UT : 3,	CONFIG : 'F U T, 0, 0, 0',
	X =  -263.697  mm,	Y =    60.088  mm,	Z =     0.001  mm,
	W =  -167.393 deg,	P =     0.014 deg,	R =   -87.773 deg
};
P[3304]{
   GP1:
	UF : 7, UT : 3,	CONFIG : 'F U T, 0, 1, 0',
	X =  -267.363  mm,	Y =    40.814  mm,	Z =     0.000  mm,
	W =  -167.383 deg,	P =     0.011 deg,	R =   -83.624 deg
};
P[3305]{
   GP1:
	UF : 7, UT : 3,	CONFIG : 'F U T, 0, 1, 0',
	X =  -269.616  mm,	Y =    21.277  mm,	Z =     0.000  mm,
	W =  -167.373 deg,	P =     0.007 deg,	R =   -79.483 deg
};
P[3306]{
   GP1:
	UF : 7, UT : 3,	CONFIG : 'F U T, 0, 1, 0',
	X =  -270.465  mm,	Y =     0.000  mm,	Z =     0.000  mm,
	W =  -167.363 deg,	P =     0.001 deg,	R =   -75.503 deg
};
P[3307]{
   GP1:
	UF : 7, UT : 3,	CONFIG : 'F U T, 0, 1, 0',
	X =  -270.465  mm,	Y =     0.000  mm,	Z =     0.000  mm,
	W =  -167.363 deg,	P =     0.001 deg,	R =   -75.503 deg
};
P[3308]{
   GP1:
	UF : 7, UT : 3,	CONFIG : 'F U T, 0, 1, 0',
	X =  -270.465  mm,	Y =     0.000  mm,	Z =     0.000  mm,
	W =  -167.363 deg,	P =     0.001 deg,	R =   -75.503 deg
};
P[3309]{
   GP1:
	UF : 7, UT : 3,	CONFIG : 'F U T, 0, 1, 0',
	X =  -270.465  mm,	Y =     0.000  mm,	Z =     0.000  mm,
	W =  -167.363 deg,	P =     0.001 deg,	R =   -75.503 deg
};
P[3310]{
   GP1:
	UF : 7, UT : 3,
	J1 =  -129.583 deg,	J2 =    24.319 deg,	J3 =   -28.425 deg,
	J4 =   110.695 deg,	J5 =   124.219 deg,	J6 =   -55.036 deg
};
/END
